LIN {X 0,Y 523.916,Z 196.85,A -85,B 0,C 180,E1 -4806.403,E2 -4806.403} C_VEL
LIN {X 0,Y 523.927,Z 196.844,A -85,B 0,C 180,E1 -4809.083,E2 -4809.083} C_VEL
LIN {X 0,Y 523.968,Z 196.839,A -85,B 0,C 180,E1 -4811.312,E2 -4811.312} C_VEL
LIN {X 0,Y 523.951,Z 196.84,A -85,B 0,C 180,E1 -4814.691,E2 -4814.691} C_VEL
LIN {X 0,Y 523.951,Z 196.846,A -85,B 0,C 180,E1 -4817.881,E2 -4817.881} C_VEL
LIN {X 0,Y 523.972,Z 196.843,A -85,B 0,C 180,E1 -4819.923,E2 -4819.923} C_VEL
LIN {X 0,Y 523.905,Z 196.844,A -85,B 0,C 180,E1 -4822.868,E2 -4822.868} C_VEL
LIN {X 0,Y 523.937,Z 196.847,A -85,B 0,C 180,E1 -4825.71,E2 -4825.71} C_VEL
LIN {X 0,Y 523.925,Z 196.843,A -85,B 0,C 180,E1 -4828.456,E2 -4828.456} C_VEL
LIN {X 0,Y 523.943,Z 196.841,A -85,B 0,C 180,E1 -4831.126,E2 -4831.126} C_VEL
LIN {X 0,Y 523.975,Z 196.842,A -85,B 0,C 180,E1 -4833.98,E2 -4833.98} C_VEL
LIN {X 0,Y 523.928,Z 196.842,A -85,B 0,C 180,E1 -4836.27,E2 -4836.27} C_VEL
LIN {X 0,Y 523.938,Z 196.834,A -85,B 0,C 180,E1 -4838.766,E2 -4838.766} C_VEL
LIN {X 0,Y 523.945,Z 196.843,A -85,B 0,C 180,E1 -4841.221,E2 -4841.221} C_VEL
LIN {X 0,Y 523.932,Z 196.848,A -85,B 0,C 180,E1 -4843.639,E2 -4843.639} C_VEL
LIN {X 0,Y 523.932,Z 196.844,A -85,B 0,C 180,E1 -4846.028,E2 -4846.028} C_VEL
LIN {X 0,Y 524.002,Z 196.833,A -85,B 0,C 180,E1 -4848.394,E2 -4848.394} C_VEL
LIN {X 0,Y 523.999,Z 196.84,A -85,B 0,C 180,E1 -4851.516,E2 -4851.516} C_VEL
LIN {X 0,Y 524.077,Z 196.824,A -85,B 0,C 180,E1 -4854.614,E2 -4854.614} C_VEL
LIN {X 0,Y 524.102,Z 196.826,A -85,B 0,C 180,E1 -4857.695,E2 -4857.695} C_VEL
LIN {X 0,Y 524.117,Z 196.818,A -85,B 0,C 180,E1 -4860.768,E2 -4860.768} C_VEL
LIN {X 0,Y 524.067,Z 196.83,A -85,B 0,C 180,E1 -4863.075,E2 -4863.075} C_VEL
LIN {X 0,Y 524.037,Z 196.829,A -85,B 0,C 180,E1 -4866.159,E2 -4866.159} C_VEL
LIN {X 0,Y 523.995,Z 196.84,A -85,B 0,C 180,E1 -4869.262,E2 -4869.262} C_VEL
LIN {X 0,Y 523.999,Z 196.835,A -85,B 0,C 180,E1 -4871.743,E2 -4871.743} C_VEL
LIN {X 0,Y 523.983,Z 196.843,A -85,B 0,C 180,E1 -4875.053,E2 -4875.053} C_VEL
LIN {X 0,Y 523.956,Z 196.839,A -85,B 0,C 180,E1 -4877.969,E2 -4877.969} C_VEL
LIN {X 0,Y 523.963,Z 196.838,A -85,B 0,C 180,E1 -4880.41,E2 -4880.41} C_VEL
LIN {X 0,Y 523.908,Z 196.851,A -85,B 0,C 180,E1 -4882.894,E2 -4882.894} C_VEL
LIN {X 0,Y 523.945,Z 196.835,A -85,B 0,C 180,E1 -4885.419,E2 -4885.419} C_VEL
LIN {X 0,Y 523.963,Z 196.837,A -85,B 0,C 180,E1 -4887.999,E2 -4887.999} C_VEL
LIN {X 0,Y 523.946,Z 196.847,A -85,B 0,C 180,E1 -4890.857,E2 -4890.857} C_VEL
LIN {X 0,Y 523.955,Z 196.838,A -85,B 0,C 180,E1 -4893.736,E2 -4893.736} C_VEL
LIN {X 0,Y 523.917,Z 196.846,A -85,B 0,C 180,E1 -4896.405,E2 -4896.405} C_VEL
LIN {X 0,Y 523.918,Z 196.848,A -85,B 0,C 180,E1 -4899.085,E2 -4899.085} C_VEL
LIN {X 0,Y 523.951,Z 196.839,A -85,B 0,C 180,E1 -4902.119,E2 -4902.119} C_VEL
LIN {X 0,Y 523.951,Z 196.842,A -85,B 0,C 180,E1 -4905.309,E2 -4905.309} C_VEL
LIN {X 0,Y 523.919,Z 196.851,A -85,B 0,C 180,E1 -4906.923,E2 -4906.923} C_VEL
LIN {X 0,Y 523.252,Z 196.929,A -85,B 0,C 180,E1 -4907.564,E2 -4907.564} C_VEL
LIN {X 0,Y 520.407,Z 197.288,A -85,B 0,C 180,E1 -4908.606,E2 -4908.606} C_VEL
LIN {X 0,Y 518.001,Z 197.588,A -85,B 0,C 180,E1 -4909.445,E2 -4909.445} C_VEL
LIN {X 0,Y 516.964,Z 197.715,A -85,B 0,C 180,E1 -4910.093,E2 -4910.093} C_VEL
LIN {X 0,Y 516.878,Z 197.725,A -85,B 0,C 180,E1 -4910.312,E2 -4910.312} C_VEL
LIN {X 0,Y 516.874,Z 197.722,A -85,B 0,C 180,E1 -4913.344,E2 -4913.344} C_VEL
LIN {X 0,Y 516.905,Z 197.721,A -85,B 0,C 180,E1 -4916.121,E2 -4916.121} C_VEL
LIN {X 0,Y 516.89,Z 197.725,A -85,B 0,C 180,E1 -4918.936,E2 -4918.936} C_VEL
LIN {X 0,Y 516.918,Z 197.719,A -85,B 0,C 180,E1 -4921.585,E2 -4921.585} C_VEL
LIN {X 0,Y 516.91,Z 197.725,A -85,B 0,C 180,E1 -4924.642,E2 -4924.642} C_VEL
LIN {X 0,Y 516.927,Z 197.807,A -85,B 0,C 180,E1 -4924.939,E2 -4924.939} C_VEL
LIN {X 0,Y 519.115,Z 207.96,A -85,B 0,C 180,E1 -4926.672,E2 -4926.672} C_VEL
LIN {X 0,Y 518.935,Z 218.424,A -85,B 0,C 180,E1 -4928.27,E2 -4928.27} C_VEL
LIN {X 0,Y 521.961,Z 232.108,A -85,B 0,C 180,E1 -4928.602,E2 -4928.602} C_VEL
LIN {X 0,Y 520.964,Z 381.412,A -85,B 0,C 180,E1 -4930.729,E2 -4930.729} C_VEL
LIN {X 0,Y 520.722,Z 395.433,A -85,B 0,C 180,E1 -4931.049,E2 -4931.049} C_VEL
LIN {X 0,Y 520.379,Z 409.153,A -85,B 0,C 180,E1 -4931.496,E2 -4931.496} C_VEL
LIN {X 0,Y 519.89,Z 422.978,A -85,B 0,C 180,E1 -4932.089,E2 -4932.089} C_VEL
LIN {X 0,Y 519.503,Z 435.806,A -85,B 0,C 180,E1 -4932.787,E2 -4932.787} C_VEL
LIN {X 0,Y 518.969,Z 449.181,A -85,B 0,C 180,E1 -4933.681,E2 -4933.681} C_VEL
LIN {X 0,Y 518.45,Z 461.571,A -85,B 0,C 180,E1 -4934.687,E2 -4934.687} C_VEL
LIN {X 0,Y 517.921,Z 473.611,A -85,B 0,C 180,E1 -4935.863,E2 -4935.863} C_VEL
LIN {X 0,Y 517.492,Z 483.799,A -85,B 0,C 180,E1 -4937.051,E2 -4937.051} C_VEL
LIN {X 0,Y 517.082,Z 493.77,A -85,B 0,C 180,E1 -4938.435,E2 -4938.435} C_VEL
LIN {X 0,Y 516.807,Z 502.039,A -85,B 0,C 180,E1 -4939.818,E2 -4939.818} C_VEL
LIN {X 0,Y 516.575,Z 509.804,A -85,B 0,C 180,E1 -4941.393,E2 -4941.393} C_VEL
LIN {X 0,Y 516.408,Z 515.988,A -85,B 0,C 180,E1 -4942.965,E2 -4942.965} C_VEL
LIN {X 0,Y 516.383,Z 520.763,A -85,B 0,C 180,E1 -4944.533,E2 -4944.533} C_VEL
LIN {X 0,Y 516.326,Z 524.265,A -85,B 0,C 180,E1 -4946.098,E2 -4946.098} C_VEL
LIN {X 0,Y 516.259,Z 526.586,A -85,B 0,C 180,E1 -4947.659,E2 -4947.659} C_VEL
LIN {X 0,Y 516.156,Z 527.776,A -85,B 0,C 180,E1 -4949.22,E2 -4949.22} C_VEL
LIN {X 0,Y 516.157,Z 527.795,A -85,B 0,C 180,E1 -4950.78,E2 -4950.78} C_VEL
LIN {X 0,Y 516.259,Z 526.681,A -85,B 0,C 180,E1 -4952.341,E2 -4952.341} C_VEL
LIN {X 0,Y 516.326,Z 524.436,A -85,B 0,C 180,E1 -4953.902,E2 -4953.902} C_VEL
LIN {X 0,Y 516.379,Z 521.005,A -85,B 0,C 180,E1 -4955.467,E2 -4955.467} C_VEL
LIN {X 0,Y 516.407,Z 516.308,A -85,B 0,C 180,E1 -4957.035,E2 -4957.035} C_VEL
LIN {X 0,Y 516.573,Z 510.218,A -85,B 0,C 180,E1 -4958.607,E2 -4958.607} C_VEL
LIN {X 0,Y 516.802,Z 502.549,A -85,B 0,C 180,E1 -4960.182,E2 -4960.182} C_VEL
LIN {X 0,Y 517.064,Z 494.37,A -85,B 0,C 180,E1 -4961.565,E2 -4961.565} C_VEL
LIN {X 0,Y 517.453,Z 484.518,A -85,B 0,C 180,E1 -4962.95,E2 -4962.95} C_VEL
LIN {X 0,Y 517.887,Z 474.412,A -85,B 0,C 180,E1 -4964.138,E2 -4964.138} C_VEL
LIN {X 0,Y 518.366,Z 462.579,A -85,B 0,C 180,E1 -4965.311,E2 -4965.311} C_VEL
LIN {X 0,Y 518.917,Z 450.576,A -85,B 0,C 180,E1 -4966.301,E2 -4966.301} C_VEL
LIN {X 0,Y 519.386,Z 438.788,A -85,B 0,C 180,E1 -4967.116,E2 -4967.116} C_VEL
LIN {X 0,Y 519.863,Z 424.732,A -85,B 0,C 180,E1 -4967.912,E2 -4967.912} C_VEL
LIN {X 0,Y 520.353,Z 410.13,A -85,B 0,C 180,E1 -4968.556,E2 -4968.556} C_VEL
LIN {X 0,Y 520.665,Z 394.698,A -85,B 0,C 180,E1 -4969.063,E2 -4969.063} C_VEL
LIN {X 0,Y 520.953,Z 379.884,A -85,B 0,C 180,E1 -4969.388,E2 -4969.388} C_VEL
LIN {X 0,Y 521.999,Z 232.476,A -85,B 0,C 180,E1 -4971.481,E2 -4971.481} C_VEL
LIN {X 0,Y 518.886,Z 218.209,A -85,B 0,C 180,E1 -4971.828,E2 -4971.828} C_VEL
LIN {X 0,Y 519.197,Z 208.527,A -85,B 0,C 180,E1 -4973.324,E2 -4973.324} C_VEL
LIN {X 0,Y 516.932,Z 197.723,A -85,B 0,C 180,E1 -4975.195,E2 -4975.195} C_VEL
LIN {X 0,Y 516.926,Z 197.722,A -85,B 0,C 180,E1 -4977.905,E2 -4977.905} C_VEL
LIN {X 0,Y 516.891,Z 197.722,A -85,B 0,C 180,E1 -4980.203,E2 -4980.203} C_VEL
LIN {X 0,Y 516.895,Z 197.723,A -85,B 0,C 180,E1 -4982.946,E2 -4982.946} C_VEL
LIN {X 0,Y 516.884,Z 197.725,A -85,B 0,C 180,E1 -4985.778,E2 -4985.778} C_VEL
LIN {X 0,Y 516.879,Z 197.724,A -85,B 0,C 180,E1 -4988.715,E2 -4988.715} C_VEL
LIN {X 0,Y 516.912,Z 197.72,A -85,B 0,C 180,E1 -4991.774,E2 -4991.774} C_VEL
LIN {X 0,Y 516.918,Z 197.72,A -85,B 0,C 180,E1 -4995.009,E2 -4995.009} C_VEL
LIN {X 0,Y 516.917,Z 197.713,A -85,B 0,C 180,E1 -4998.397,E2 -4998.397} C_VEL
LIN {X 0,Y 516.877,Z 197.724,A -85,B 0,C 180,E1 -5001.284,E2 -5001.284} C_VEL
LIN {X 0,Y 516.885,Z 197.719,A -85,B 0,C 180,E1 -5004.221,E2 -5004.221} C_VEL
LIN {X 0,Y 516.891,Z 197.723,A -85,B 0,C 180,E1 -5007.053,E2 -5007.053} C_VEL
LIN {X 0,Y 516.895,Z 197.717,A -85,B 0,C 180,E1 -5009.796,E2 -5009.796} C_VEL
LIN {X 0,Y 516.921,Z 197.717,A -85,B 0,C 180,E1 -5012.467,E2 -5012.467} C_VEL
LIN {X 0,Y 516.902,Z 197.726,A -85,B 0,C 180,E1 -5015.071,E2 -5015.071} C_VEL
LIN {X 0,Y 516.878,Z 197.722,A -85,B 0,C 180,E1 -5018.462,E2 -5018.462} C_VEL
LIN {X 0,Y 516.897,Z 197.724,A -85,B 0,C 180,E1 -5020.955,E2 -5020.955} C_VEL
LIN {X 0,Y 516.909,Z 197.719,A -85,B 0,C 180,E1 -5023.41,E2 -5023.41} C_VEL
LIN {X 0,Y 516.886,Z 197.717,A -85,B 0,C 180,E1 -5025.833,E2 -5025.833} C_VEL
LIN {X 0,Y 516.956,Z 197.713,A -85,B 0,C 180,E1 -5028.233,E2 -5028.233} C_VEL
LIN {X 0,Y 516.961,Z 197.712,A -85,B 0,C 180,E1 -5031.399,E2 -5031.399} C_VEL
LIN {X 0,Y 517.001,Z 197.704,A -85,B 0,C 180,E1 -5033.757,E2 -5033.757} C_VEL
LIN {X 0,Y 517.007,Z 197.711,A -85,B 0,C 180,E1 -5036.883,E2 -5036.883} C_VEL
LIN {X 0,Y 517.073,Z 197.695,A -85,B 0,C 180,E1 -5040,E2 -5040} C_VEL
LIN {X 0,Y 517.008,Z 197.705,A -85,B 0,C 180,E1 -5043.117,E2 -5043.117} C_VEL
LIN {X 0,Y 517,Z 197.71,A -85,B 0,C 180,E1 -5046.243,E2 -5046.243} C_VEL
LIN {X 0,Y 516.949,Z 197.711,A -85,B 0,C 180,E1 -5049.389,E2 -5049.389} C_VEL
LIN {X 0,Y 516.947,Z 197.713,A -85,B 0,C 180,E1 -5051.81,E2 -5051.81} C_VEL
LIN {X 0,Y 516.937,Z 197.715,A -85,B 0,C 180,E1 -5055.148,E2 -5055.148} C_VEL
LIN {X 0,Y 516.917,Z 197.72,A -85,B 0,C 180,E1 -5058.222,E2 -5058.222} C_VEL
LIN {X 0,Y 516.904,Z 197.72,A -85,B 0,C 180,E1 -5060.702,E2 -5060.702} C_VEL
LIN {X 0,Y 516.902,Z 197.724,A -85,B 0,C 180,E1 -5064.072,E2 -5064.072} C_VEL
LIN {X 0,Y 516.918,Z 197.72,A -85,B 0,C 180,E1 -5066.658,E2 -5066.658} C_VEL
LIN {X 0,Y 516.917,Z 197.717,A -85,B 0,C 180,E1 -5069.527,E2 -5069.527} C_VEL
LIN {X 0,Y 516.893,Z 197.721,A -85,B 0,C 180,E1 -5072.545,E2 -5072.545} C_VEL
LIN {X 0,Y 516.876,Z 197.721,A -85,B 0,C 180,E1 -5075.333,E2 -5075.333} C_VEL
LIN {X 0,Y 516.874,Z 197.727,A -85,B 0,C 180,E1 -5077.944,E2 -5077.944} C_VEL
LIN {X 0,Y 516.879,Z 197.717,A -85,B 0,C 180,E1 -5080.742,E2 -5080.742} C_VEL
LIN {X 0,Y 516.878,Z 197.722,A -85,B 0,C 180,E1 -5082.832,E2 -5082.832} C_VEL
LIN {X 0,Y 516.917,Z 197.717,A -85,B 0,C 180,E1 -5085.011,E2 -5085.011} C_VEL
LIN {X 0,Y 516.918,Z 197.719,A -85,B 0,C 180,E1 -5088.398,E2 -5088.398} C_VEL
LIN {X 0,Y 516.882,Z 197.722,A -85,B 0,C 180,E1 -5091.285,E2 -5091.285} C_VEL
LIN {X 0,Y 516.884,Z 197.726,A -85,B 0,C 180,E1 -5094.222,E2 -5094.222} C_VEL
LIN {X 0,Y 516.893,Z 197.721,A -85,B 0,C 180,E1 -5097.054,E2 -5097.054} C_VEL
LIN {X 0,Y 516.889,Z 197.727,A -85,B 0,C 180,E1 -5099.797,E2 -5099.797} C_VEL
LIN {X 0,Y 516.942,Z 197.766,A -85,B 0,C 180,E1 -5101.726,E2 -5101.726} C_VEL
LIN {X 0,Y 519.956,Z 211.044,A -85,B 0,C 180,E1 -5103.727,E2 -5103.727} C_VEL
LIN {X 0,Y 519.317,Z 231.522,A -85,B 0,C 180,E1 -5106.471,E2 -5106.471} C_VEL
LIN {X 0,Y 518.882,Z 244.581,A -85,B 0,C 180,E1 -5108.199,E2 -5108.199} C_VEL
LIN {X 0,Y 521.857,Z 259.942,A -85,B 0,C 180,E1 -5108.558,E2 -5108.558} C_VEL
LIN {X 0,Y 520.958,Z 393.454,A -85,B 0,C 180,E1 -5110.442,E2 -5110.442} C_VEL
LIN {X 0,Y 520.783,Z 413.905,A -85,B 0,C 180,E1 -5110.772,E2 -5110.772} C_VEL
LIN {X 0,Y 520.463,Z 428.98,A -85,B 0,C 180,E1 -5111.167,E2 -5111.167} C_VEL
LIN {X 0,Y 520.064,Z 443.174,A -85,B 0,C 180,E1 -5111.688,E2 -5111.688} C_VEL
LIN {X 0,Y 519.498,Z 457.644,A -85,B 0,C 180,E1 -5112.381,E2 -5112.381} C_VEL
LIN {X 0,Y 519.055,Z 470.865,A -85,B 0,C 180,E1 -5113.177,E2 -5113.177} C_VEL
LIN {X 0,Y 518.569,Z 483.587,A -85,B 0,C 180,E1 -5114.11,E2 -5114.11} C_VEL
LIN {X 0,Y 517.958,Z 496.586,A -85,B 0,C 180,E1 -5115.262,E2 -5115.262} C_VEL
LIN {X 0,Y 517.529,Z 507.783,A -85,B 0,C 180,E1 -5116.453,E2 -5116.453} C_VEL
LIN {X 0,Y 517.131,Z 518.653,A -85,B 0,C 180,E1 -5117.84,E2 -5117.84} C_VEL
LIN {X 0,Y 516.865,Z 527.703,A -85,B 0,C 180,E1 -5119.225,E2 -5119.225} C_VEL
LIN {X 0,Y 516.575,Z 535.208,A -85,B 0,C 180,E1 -5120.604,E2 -5120.604} C_VEL
LIN {X 0,Y 516.443,Z 542.215,A -85,B 0,C 180,E1 -5122.179,E2 -5122.179} C_VEL
LIN {X 0,Y 516.36,Z 547.724,A -85,B 0,C 180,E1 -5123.749,E2 -5123.749} C_VEL
LIN {X 0,Y 516.238,Z 551.887,A -85,B 0,C 180,E1 -5125.315,E2 -5125.315} C_VEL
LIN {X 0,Y 516.271,Z 554.808,A -85,B 0,C 180,E1 -5126.879,E2 -5126.879} C_VEL
LIN {X 0,Y 516.189,Z 556.548,A -85,B 0,C 180,E1 -5128.44,E2 -5128.44} C_VEL
LIN {X 0,Y 516.151,Z 557.144,A -85,B 0,C 180,E1 -5130,E2 -5130} C_VEL
LIN {X 0,Y 516.189,Z 556.545,A -85,B 0,C 180,E1 -5131.56,E2 -5131.56} C_VEL
LIN {X 0,Y 516.271,Z 554.803,A -85,B 0,C 180,E1 -5133.121,E2 -5133.121} C_VEL
LIN {X 0,Y 516.238,Z 551.885,A -85,B 0,C 180,E1 -5134.685,E2 -5134.685} C_VEL
LIN {X 0,Y 516.375,Z 547.728,A -85,B 0,C 180,E1 -5136.251,E2 -5136.251} C_VEL
LIN {X 0,Y 516.443,Z 542.216,A -85,B 0,C 180,E1 -5137.821,E2 -5137.821} C_VEL
LIN {X 0,Y 516.575,Z 535.202,A -85,B 0,C 180,E1 -5139.396,E2 -5139.396} C_VEL
LIN {X 0,Y 516.863,Z 527.698,A -85,B 0,C 180,E1 -5140.775,E2 -5140.775} C_VEL
LIN {X 0,Y 517.097,Z 518.923,A -85,B 0,C 180,E1 -5142.121,E2 -5142.121} C_VEL
LIN {X 0,Y 517.489,Z 509.423,A -85,B 0,C 180,E1 -5143.348,E2 -5143.348} C_VEL
LIN {X 0,Y 517.917,Z 498.552,A -85,B 0,C 180,E1 -5144.539,E2 -5144.539} C_VEL
LIN {X 0,Y 518.355,Z 487.283,A -85,B 0,C 180,E1 -5145.582,E2 -5145.582} C_VEL
LIN {X 0,Y 518.912,Z 473.727,A -85,B 0,C 180,E1 -5146.625,E2 -5146.625} C_VEL
LIN {X 0,Y 519.493,Z 459.409,A -85,B 0,C 180,E1 -5147.518,E2 -5147.518} C_VEL
LIN {X 0,Y 519.957,Z 445.443,A -85,B 0,C 180,E1 -5148.214,E2 -5148.214} C_VEL
LIN {X 0,Y 520.407,Z 430.524,A -85,B 0,C 180,E1 -5148.784,E2 -5148.784} C_VEL
LIN {X 0,Y 520.758,Z 415.339,A -85,B 0,C 180,E1 -5149.197,E2 -5149.197} C_VEL
LIN {X 0,Y 520.972,Z 395.646,A -85,B 0,C 180,E1 -5149.526,E2 -5149.526} C_VEL
LIN {X 0,Y 521.861,Z 259.839,A -85,B 0,C 180,E1 -5151.443,E2 -5151.443} C_VEL
LIN {X 0,Y 518.886,Z 244.592,A -85,B 0,C 180,E1 -5151.799,E2 -5151.799} C_VEL
LIN {X 0,Y 519.653,Z 222.079,A -85,B 0,C 180,E1 -5154.787,E2 -5154.787} C_VEL
LIN {X 0,Y 519.956,Z 211.043,A -85,B 0,C 180,E1 -5156.273,E2 -5156.273} C_VEL
LIN {X 0,Y 516.919,Z 197.724,A -85,B 0,C 180,E1 -5158.31,E2 -5158.31} C_VEL
LIN {X 0,Y 516.886,Z 197.719,A -85,B 0,C 180,E1 -5161.109,E2 -5161.109} C_VEL
LIN {X 0,Y 516.908,Z 197.718,A -85,B 0,C 180,E1 -5163.966,E2 -5163.966} C_VEL
LIN {X 0,Y 516.878,Z 197.723,A -85,B 0,C 180,E1 -5166.745,E2 -5166.745} C_VEL
LIN {X 0,Y 516.899,Z 197.724,A -85,B 0,C 180,E1 -5169.719,E2 -5169.719} C_VEL
LIN {X 0,Y 516.914,Z 197.722,A -85,B 0,C 180,E1 -5171.774,E2 -5171.774} C_VEL
LIN {X 0,Y 516.917,Z 197.715,A -85,B 0,C 180,E1 -5175.009,E2 -5175.009} C_VEL
LIN {X 0,Y 516.916,Z 197.718,A -85,B 0,C 180,E1 -5178.397,E2 -5178.397} C_VEL
LIN {X 0,Y 516.88,Z 197.721,A -85,B 0,C 180,E1 -5181.284,E2 -5181.284} C_VEL
LIN {X 0,Y 516.884,Z 197.722,A -85,B 0,C 180,E1 -5184.221,E2 -5184.221} C_VEL
LIN {X 0,Y 516.89,Z 197.717,A -85,B 0,C 180,E1 -5187.053,E2 -5187.053} C_VEL
LIN {X 0,Y 516.894,Z 197.724,A -85,B 0,C 180,E1 -5189.797,E2 -5189.797} C_VEL
LIN {X 0,Y 516.92,Z 197.715,A -85,B 0,C 180,E1 -5192.467,E2 -5192.467} C_VEL
LIN {X 0,Y 516.902,Z 197.719,A -85,B 0,C 180,E1 -5195.072,E2 -5195.072} C_VEL
LIN {X 0,Y 516.878,Z 197.713,A -85,B 0,C 180,E1 -5198.462,E2 -5198.462} C_VEL
LIN {X 0,Y 516.896,Z 197.718,A -85,B 0,C 180,E1 -5200.955,E2 -5200.955} C_VEL
LIN {X 0,Y 516.909,Z 197.723,A -85,B 0,C 180,E1 -5203.41,E2 -5203.41} C_VEL
LIN {X 0,Y 516.887,Z 197.724,A -85,B 0,C 180,E1 -5205.833,E2 -5205.833} C_VEL
LIN {X 0,Y 516.948,Z 197.714,A -85,B 0,C 180,E1 -5209.028,E2 -5209.028} C_VEL
LIN {X 0,Y 516.969,Z 197.709,A -85,B 0,C 180,E1 -5212.187,E2 -5212.187} C_VEL
LIN {X 0,Y 517.024,Z 197.702,A -85,B 0,C 180,E1 -5214.54,E2 -5214.54} C_VEL
LIN {X 0,Y 517.074,Z 197.702,A -85,B 0,C 180,E1 -5217.663,E2 -5217.663} C_VEL
LIN {X 0,Y 517.087,Z 197.694,A -85,B 0,C 180,E1 -5220.779,E2 -5220.779} C_VEL
LIN {X 0,Y 517.008,Z 197.71,A -85,B 0,C 180,E1 -5223.117,E2 -5223.117} C_VEL
LIN {X 0,Y 517.001,Z 197.705,A -85,B 0,C 180,E1 -5226.243,E2 -5226.243} C_VEL
LIN {X 0,Y 516.949,Z 197.719,A -85,B 0,C 180,E1 -5229.389,E2 -5229.389} C_VEL
LIN {X 0,Y 516.948,Z 197.712,A -85,B 0,C 180,E1 -5231.811,E2 -5231.811} C_VEL
LIN {X 0,Y 516.935,Z 197.722,A -85,B 0,C 180,E1 -5235.147,E2 -5235.147} C_VEL
LIN {X 0,Y 516.917,Z 197.716,A -85,B 0,C 180,E1 -5238.223,E2 -5238.223} C_VEL
LIN {X 0,Y 516.904,Z 197.72,A -85,B 0,C 180,E1 -5240.702,E2 -5240.702} C_VEL
LIN {X 0,Y 516.903,Z 197.716,A -85,B 0,C 180,E1 -5244.073,E2 -5244.073} C_VEL
LIN {X 0,Y 516.919,Z 197.71,A -85,B 0,C 180,E1 -5246.658,E2 -5246.658} C_VEL
LIN {X 0,Y 516.918,Z 197.718,A -85,B 0,C 180,E1 -5249.527,E2 -5249.527} C_VEL
LIN {X 0,Y 516.894,Z 197.722,A -85,B 0,C 180,E1 -5252.545,E2 -5252.545} C_VEL
LIN {X 0,Y 516.877,Z 197.724,A -85,B 0,C 180,E1 -5255.333,E2 -5255.333} C_VEL
LIN {X 0,Y 516.876,Z 197.72,A -85,B 0,C 180,E1 -5257.944,E2 -5257.944} C_VEL
LIN {X 0,Y 516.88,Z 197.727,A -85,B 0,C 180,E1 -5260.742,E2 -5260.742} C_VEL
LIN {X 0,Y 516.898,Z 197.726,A -85,B 0,C 180,E1 -5262.83,E2 -5262.83} C_VEL
LIN {X 0,Y 516.918,Z 197.721,A -85,B 0,C 180,E1 -5265.011,E2 -5265.011} C_VEL
LIN {X 0,Y 516.913,Z 197.721,A -85,B 0,C 180,E1 -5268.399,E2 -5268.399} C_VEL
LIN {X 0,Y 516.878,Z 197.725,A -85,B 0,C 180,E1 -5270.312,E2 -5270.312} C_VEL
LIN {X 0,Y 516.207,Z 197.808,A -85,B 0,C 180,E1 -5270.962,E2 -5270.962} C_VEL
LIN {X 0,Y 513.36,Z 198.16,A -85,B 0,C 180,E1 -5272.018,E2 -5272.018} C_VEL
LIN {X 0,Y 510.949,Z 198.466,A -85,B 0,C 180,E1 -5272.868,E2 -5272.868} C_VEL
LIN {X 0,Y 509.906,Z 198.59,A -85,B 0,C 180,E1 -5273.525,E2 -5273.525} C_VEL
LIN {X 0,Y 509.817,Z 198.6,A -85,B 0,C 180,E1 -5273.747,E2 -5273.747} C_VEL
LIN {X 0,Y 509.857,Z 198.601,A -85,B 0,C 180,E1 -5276.54,E2 -5276.54} C_VEL
LIN {X 0,Y 509.844,Z 198.601,A -85,B 0,C 180,E1 -5279.335,E2 -5279.335} C_VEL
LIN {X 0,Y 509.893,Z 198.597,A -85,B 0,C 180,E1 -5282.055,E2 -5282.055} C_VEL
LIN {X 0,Y 509.872,Z 198.661,A -85,B 0,C 180,E1 -5284.677,E2 -5284.677} C_VEL
LIN {X 0,Y 512.223,Z 209.489,A -85,B 0,C 180,E1 -5286.554,E2 -5286.554} C_VEL
LIN {X 0,Y 512.076,Z 218.377,A -85,B 0,C 180,E1 -5287.952,E2 -5287.952} C_VEL
LIN {X 0,Y 515.356,Z 232.894,A -85,B 0,C 180,E1 -5288.322,E2 -5288.322} C_VEL
LIN {X 0,Y 514.284,Z 379.059,A -85,B 0,C 180,E1 -5290.423,E2 -5290.423} C_VEL
LIN {X 0,Y 514.013,Z 394.613,A -85,B 0,C 180,E1 -5290.762,E2 -5290.762} C_VEL
LIN {X 0,Y 513.657,Z 409.37,A -85,B 0,C 180,E1 -5291.245,E2 -5291.245} C_VEL
LIN {X 0,Y 513.127,Z 423.191,A -85,B 0,C 180,E1 -5291.845,E2 -5291.845} C_VEL
LIN {X 0,Y 512.724,Z 436.017,A -85,B 0,C 180,E1 -5292.552,E2 -5292.552} C_VEL
LIN {X 0,Y 512.126,Z 449.391,A -85,B 0,C 180,E1 -5293.456,E2 -5293.456} C_VEL
LIN {X 0,Y 511.566,Z 462.071,A -85,B 0,C 180,E1 -5294.502,E2 -5294.502} C_VEL
LIN {X 0,Y 510.985,Z 473.82,A -85,B 0,C 180,E1 -5295.667,E2 -5295.667} C_VEL
LIN {X 0,Y 510.552,Z 484.006,A -85,B 0,C 180,E1 -5296.872,E2 -5296.872} C_VEL
LIN {X 0,Y 510.07,Z 494.421,A -85,B 0,C 180,E1 -5298.341,E2 -5298.341} C_VEL
LIN {X 0,Y 509.743,Z 503.337,A -85,B 0,C 180,E1 -5299.876,E2 -5299.876} C_VEL
LIN {X 0,Y 509.515,Z 510.009,A -85,B 0,C 180,E1 -5301.273,E2 -5301.273} C_VEL
LIN {X 0,Y 509.356,Z 516.191,A -85,B 0,C 180,E1 -5302.867,E2 -5302.867} C_VEL
LIN {X 0,Y 509.323,Z 520.965,A -85,B 0,C 180,E1 -5304.457,E2 -5304.457} C_VEL
LIN {X 0,Y 509.252,Z 524.467,A -85,B 0,C 180,E1 -5306.043,E2 -5306.043} C_VEL
LIN {X 0,Y 509.187,Z 526.786,A -85,B 0,C 180,E1 -5307.627,E2 -5307.627} C_VEL
LIN {X 0,Y 509.07,Z 527.977,A -85,B 0,C 180,E1 -5309.209,E2 -5309.209} C_VEL
LIN {X 0,Y 509.071,Z 527.996,A -85,B 0,C 180,E1 -5310.791,E2 -5310.791} C_VEL
LIN {X 0,Y 509.188,Z 526.881,A -85,B 0,C 180,E1 -5312.373,E2 -5312.373} C_VEL
LIN {X 0,Y 509.252,Z 524.635,A -85,B 0,C 180,E1 -5313.957,E2 -5313.957} C_VEL
LIN {X 0,Y 509.317,Z 521.204,A -85,B 0,C 180,E1 -5315.543,E2 -5315.543} C_VEL
LIN {X 0,Y 509.356,Z 516.506,A -85,B 0,C 180,E1 -5317.133,E2 -5317.133} C_VEL
LIN {X 0,Y 509.513,Z 510.417,A -85,B 0,C 180,E1 -5318.727,E2 -5318.727} C_VEL
LIN {X 0,Y 509.788,Z 502.747,A -85,B 0,C 180,E1 -5320.324,E2 -5320.324} C_VEL
LIN {X 0,Y 510.064,Z 494.159,A -85,B 0,C 180,E1 -5321.789,E2 -5321.789} C_VEL
LIN {X 0,Y 510.524,Z 484.714,A -85,B 0,C 180,E1 -5323.129,E2 -5323.129} C_VEL
LIN {X 0,Y 510.973,Z 474.608,A -85,B 0,C 180,E1 -5324.334,E2 -5324.334} C_VEL
LIN {X 0,Y 511.489,Z 463.047,A -85,B 0,C 180,E1 -5325.496,E2 -5325.496} C_VEL
LIN {X 0,Y 512.09,Z 450.515,A -85,B 0,C 180,E1 -5326.545,E2 -5326.545} C_VEL
LIN {X 0,Y 512.695,Z 437.402,A -85,B 0,C 180,E1 -5327.449,E2 -5327.449} C_VEL
LIN {X 0,Y 513.108,Z 424.921,A -85,B 0,C 180,E1 -5328.156,E2 -5328.156} C_VEL
LIN {X 0,Y 513.625,Z 410.315,A -85,B 0,C 180,E1 -5328.808,E2 -5328.808} C_VEL
LIN {X 0,Y 513.97,Z 394.993,A -85,B 0,C 180,E1 -5329.318,E2 -5329.318} C_VEL
LIN {X 0,Y 514.285,Z 379.346,A -85,B 0,C 180,E1 -5329.662,E2 -5329.662} C_VEL
LIN {X 0,Y 515.341,Z 232.959,A -85,B 0,C 180,E1 -5331.767,E2 -5331.767} C_VEL
LIN {X 0,Y 512.076,Z 218.337,A -85,B 0,C 180,E1 -5332.143,E2 -5332.143} C_VEL
LIN {X 0,Y 512.323,Z 210.046,A -85,B 0,C 180,E1 -5333.441,E2 -5333.441} C_VEL
LIN {X 0,Y 509.869,Z 198.603,A -85,B 0,C 180,E1 -5335.46,E2 -5335.46} C_VEL
LIN {X 0,Y 509.897,Z 198.596,A -85,B 0,C 180,E1 -5338.1,E2 -5338.1} C_VEL
LIN {X 0,Y 509.844,Z 198.605,A -85,B 0,C 180,E1 -5341.279,E2 -5341.279} C_VEL
LIN {X 0,Y 509.858,Z 198.598,A -85,B 0,C 180,E1 -5344.202,E2 -5344.202} C_VEL
LIN {X 0,Y 509.816,Z 198.607,A -85,B 0,C 180,E1 -5347.34,E2 -5347.34} C_VEL
LIN {X 0,Y 509.835,Z 198.598,A -85,B 0,C 180,E1 -5350.381,E2 -5350.381} C_VEL
LIN {X 0,Y 509.836,Z 198.603,A -85,B 0,C 180,E1 -5353.064,E2 -5353.064} C_VEL
LIN {X 0,Y 509.826,Z 198.601,A -85,B 0,C 180,E1 -5355.792,E2 -5355.792} C_VEL
LIN {X 0,Y 509.86,Z 198.593,A -85,B 0,C 180,E1 -5358.575,E2 -5358.575} C_VEL
LIN {X 0,Y 509.846,Z 198.593,A -85,B 0,C 180,E1 -5361.786,E2 -5361.786} C_VEL
LIN {X 0,Y 509.84,Z 198.598,A -85,B 0,C 180,E1 -5364.623,E2 -5364.623} C_VEL
LIN {X 0,Y 509.859,Z 198.592,A -85,B 0,C 180,E1 -5367.481,E2 -5367.481} C_VEL
LIN {X 0,Y 509.875,Z 198.591,A -85,B 0,C 180,E1 -5370.268,E2 -5370.268} C_VEL
LIN {X 0,Y 509.878,Z 198.6,A -85,B 0,C 180,E1 -5372.944,E2 -5372.944} C_VEL
LIN {X 0,Y 509.861,Z 198.597,A -85,B 0,C 180,E1 -5375.573,E2 -5375.573} C_VEL
LIN {X 0,Y 509.842,Z 198.606,A -85,B 0,C 180,E1 -5378.998,E2 -5378.998} C_VEL
LIN {X 0,Y 509.88,Z 198.59,A -85,B 0,C 180,E1 -5381.999,E2 -5381.999} C_VEL
LIN {X 0,Y 509.901,Z 198.597,A -85,B 0,C 180,E1 -5384.818,E2 -5384.818} C_VEL
LIN {X 0,Y 509.897,Z 198.591,A -85,B 0,C 180,E1 -5388.12,E2 -5388.12} C_VEL
LIN {X 0,Y 509.908,Z 198.591,A -85,B 0,C 180,E1 -5391.28,E2 -5391.28} C_VEL
LIN {X 0,Y 509.969,Z 198.58,A -85,B 0,C 180,E1 -5393.67,E2 -5393.67} C_VEL
LIN {X 0,Y 510.045,Z 198.572,A -85,B 0,C 180,E1 -5397.631,E2 -5397.631} C_VEL
LIN {X 0,Y 510.057,Z 198.578,A -85,B 0,C 180,E1 -5400.789,E2 -5400.789} C_VEL
LIN {X 0,Y 509.95,Z 198.583,A -85,B 0,C 180,E1 -5403.16,E2 -5403.16} C_VEL
LIN {X 0,Y 509.969,Z 198.587,A -85,B 0,C 180,E1 -5406.33,E2 -5406.33} C_VEL
LIN {X 0,Y 509.909,Z 198.594,A -85,B 0,C 180,E1 -5408.72,E2 -5408.72} C_VEL
LIN {X 0,Y 509.895,Z 198.593,A -85,B 0,C 180,E1 -5411.932,E2 -5411.932} C_VEL
LIN {X 0,Y 509.884,Z 198.594,A -85,B 0,C 180,E1 -5415.242,E2 -5415.242} C_VEL
LIN {X 0,Y 509.879,Z 198.593,A -85,B 0,C 180,E1 -5418.001,E2 -5418.001} C_VEL
LIN {X 0,Y 509.842,Z 198.597,A -85,B 0,C 180,E1 -5421.002,E2 -5421.002} C_VEL
LIN {X 0,Y 509.828,Z 198.601,A -85,B 0,C 180,E1 -5423.563,E2 -5423.563} C_VEL
LIN {X 0,Y 509.903,Z 198.597,A -85,B 0,C 180,E1 -5426.379,E2 -5426.379} C_VEL
LIN {X 0,Y 509.877,Z 198.595,A -85,B 0,C 180,E1 -5428.844,E2 -5428.844} C_VEL
LIN {X 0,Y 509.819,Z 198.602,A -85,B 0,C 180,E1 -5431.59,E2 -5431.59} C_VEL
LIN {X 0,Y 509.846,Z 198.602,A -85,B 0,C 180,E1 -5434.414,E2 -5434.414} C_VEL
LIN {X 0,Y 509.812,Z 198.601,A -85,B 0,C 180,E1 -5437.341,E2 -5437.341} C_VEL
LIN {X 0,Y 509.832,Z 198.596,A -85,B 0,C 180,E1 -5440.383,E2 -5440.383} C_VEL
LIN {X 0,Y 509.818,Z 198.601,A -85,B 0,C 180,E1 -5443.063,E2 -5443.063} C_VEL
LIN {X 0,Y 509.825,Z 198.606,A -85,B 0,C 180,E1 -5445.793,E2 -5445.793} C_VEL
LIN {X 0,Y 509.861,Z 198.597,A -85,B 0,C 180,E1 -5448.576,E2 -5448.576} C_VEL
LIN {X 0,Y 509.848,Z 198.602,A -85,B 0,C 180,E1 -5451.787,E2 -5451.787} C_VEL
LIN {X 0,Y 509.839,Z 198.6,A -85,B 0,C 180,E1 -5454.624,E2 -5454.624} C_VEL
LIN {X 0,Y 509.86,Z 198.601,A -85,B 0,C 180,E1 -5457.482,E2 -5457.482} C_VEL
LIN {X 0,Y 509.856,Z 198.603,A -85,B 0,C 180,E1 -5460.274,E2 -5460.274} C_VEL
LIN {X 0,Y 509.873,Z 198.602,A -85,B 0,C 180,E1 -5461.445,E2 -5461.445} C_VEL
LIN {X 0,Y 513.079,Z 212.434,A -85,B 0,C 180,E1 -5463.566,E2 -5463.566} C_VEL
LIN {X 0,Y 512.574,Z 229.761,A -85,B 0,C 180,E1 -5465.927,E2 -5465.927} C_VEL
LIN {X 0,Y 512.037,Z 244.433,A -85,B 0,C 180,E1 -5467.9,E2 -5467.9} C_VEL
LIN {X 0,Y 515.302,Z 261.598,A -85,B 0,C 180,E1 -5468.299,E2 -5468.299} C_VEL
LIN {X 0,Y 514.168,Z 410.043,A -85,B 0,C 180,E1 -5470.436,E2 -5470.436} C_VEL
LIN {X 0,Y 513.786,Z 425.612,A -85,B 0,C 180,E1 -5470.809,E2 -5470.809} C_VEL
LIN {X 0,Y 513.381,Z 440.605,A -85,B 0,C 180,E1 -5471.338,E2 -5471.338} C_VEL
LIN {X 0,Y 512.783,Z 455.626,A -85,B 0,C 180,E1 -5472.039,E2 -5472.039} C_VEL
LIN {X 0,Y 512.284,Z 469.143,A -85,B 0,C 180,E1 -5472.845,E2 -5472.845} C_VEL
LIN {X 0,Y 511.712,Z 481.607,A -85,B 0,C 180,E1 -5473.75,E2 -5473.75} C_VEL
LIN {X 0,Y 511.157,Z 494.287,A -85,B 0,C 180,E1 -5474.857,E2 -5474.857} C_VEL
LIN {X 0,Y 510.639,Z 505.808,A -85,B 0,C 180,E1 -5476.063,E2 -5476.063} C_VEL
LIN {X 0,Y 510.21,Z 515.508,A -85,B 0,C 180,E1 -5477.268,E2 -5477.268} C_VEL
LIN {X 0,Y 509.846,Z 525.192,A -85,B 0,C 180,E1 -5478.697,E2 -5478.697} C_VEL
LIN {X 0,Y 509.565,Z 532.975,A -85,B 0,C 180,E1 -5480.073,E2 -5480.073} C_VEL
LIN {X 0,Y 509.394,Z 540.389,A -85,B 0,C 180,E1 -5481.671,E2 -5481.671} C_VEL
LIN {X 0,Y 509.289,Z 546.271,A -85,B 0,C 180,E1 -5483.264,E2 -5483.264} C_VEL
LIN {X 0,Y 509.263,Z 549.766,A -85,B 0,C 180,E1 -5484.457,E2 -5484.457} C_VEL
LIN {X 0,Y 509.171,Z 553.298,A -85,B 0,C 180,E1 -5486.043,E2 -5486.043} C_VEL
LIN {X 0,Y 509.187,Z 555.622,A -85,B 0,C 180,E1 -5487.627,E2 -5487.627} C_VEL
LIN {X 0,Y 509.071,Z 556.789,A -85,B 0,C 180,E1 -5489.209,E2 -5489.209} C_VEL
LIN {X 0,Y 509.071,Z 556.788,A -85,B 0,C 180,E1 -5490.791,E2 -5490.791} C_VEL
LIN {X 0,Y 509.187,Z 555.618,A -85,B 0,C 180,E1 -5492.373,E2 -5492.373} C_VEL
LIN {X 0,Y 509.171,Z 553.293,A -85,B 0,C 180,E1 -5493.957,E2 -5493.957} C_VEL
LIN {X 0,Y 509.264,Z 549.768,A -85,B 0,C 180,E1 -5495.543,E2 -5495.543} C_VEL
LIN {X 0,Y 509.316,Z 544.948,A -85,B 0,C 180,E1 -5497.134,E2 -5497.134} C_VEL
LIN {X 0,Y 509.453,Z 538.706,A -85,B 0,C 180,E1 -5498.728,E2 -5498.728} C_VEL
LIN {X 0,Y 509.7,Z 530.868,A -85,B 0,C 180,E1 -5500.326,E2 -5500.326} C_VEL
LIN {X 0,Y 509.957,Z 522.391,A -85,B 0,C 180,E1 -5501.749,E2 -5501.749} C_VEL
LIN {X 0,Y 510.343,Z 512.493,A -85,B 0,C 180,E1 -5503.133,E2 -5503.133} C_VEL
LIN {X 0,Y 510.78,Z 502.225,A -85,B 0,C 180,E1 -5504.339,E2 -5504.339} C_VEL
LIN {X 0,Y 511.369,Z 489.426,A -85,B 0,C 180,E1 -5505.597,E2 -5505.597} C_VEL
LIN {X 0,Y 511.976,Z 476.39,A -85,B 0,C 180,E1 -5506.651,E2 -5506.651} C_VEL
LIN {X 0,Y 512.569,Z 462.749,A -85,B 0,C 180,E1 -5507.556,E2 -5507.556} C_VEL
LIN {X 0,Y 513.104,Z 448.626,A -85,B 0,C 180,E1 -5508.311,E2 -5508.311} C_VEL
LIN {X 0,Y 513.563,Z 434.138,A -85,B 0,C 180,E1 -5508.913,E2 -5508.913} C_VEL
LIN {X 0,Y 513.934,Z 418.679,A -85,B 0,C 180,E1 -5509.381,E2 -5509.381} C_VEL
LIN {X 0,Y 514.251,Z 402.339,A -85,B 0,C 180,E1 -5509.692,E2 -5509.692} C_VEL
LIN {X 0,Y 515.302,Z 261.597,A -85,B 0,C 180,E1 -5511.701,E2 -5511.701} C_VEL
LIN {X 0,Y 512.003,Z 244.408,A -85,B 0,C 180,E1 -5512.105,E2 -5512.105} C_VEL
LIN {X 0,Y 512.806,Z 223.461,A -85,B 0,C 180,E1 -5514.924,E2 -5514.924} C_VEL
LIN {X 0,Y 513.063,Z 212.429,A -85,B 0,C 180,E1 -5516.435,E2 -5516.435} C_VEL
LIN {X 0,Y 509.895,Z 198.598,A -85,B 0,C 180,E1 -5518.554,E2 -5518.554} C_VEL
LIN {X 0,Y 509.818,Z 198.601,A -85,B 0,C 180,E1 -5521.589,E2 -5521.589} C_VEL
LIN {X 0,Y 509.848,Z 198.6,A -85,B 0,C 180,E1 -5524.413,E2 -5524.413} C_VEL
LIN {X 0,Y 509.815,Z 198.602,A -85,B 0,C 180,E1 -5527.34,E2 -5527.34} C_VEL
LIN {X 0,Y 509.857,Z 198.6,A -85,B 0,C 180,E1 -5530.379,E2 -5530.379} C_VEL
LIN {X 0,Y 509.819,Z 198.6,A -85,B 0,C 180,E1 -5533.062,E2 -5533.062} C_VEL
LIN {X 0,Y 509.825,Z 198.604,A -85,B 0,C 180,E1 -5535.792,E2 -5535.792} C_VEL
LIN {X 0,Y 509.859,Z 198.595,A -85,B 0,C 180,E1 -5538.575,E2 -5538.575} C_VEL
LIN {X 0,Y 509.846,Z 198.602,A -85,B 0,C 180,E1 -5541.786,E2 -5541.786} C_VEL
LIN {X 0,Y 509.839,Z 198.596,A -85,B 0,C 180,E1 -5544.623,E2 -5544.623} C_VEL
LIN {X 0,Y 509.858,Z 198.597,A -85,B 0,C 180,E1 -5547.481,E2 -5547.481} C_VEL
LIN {X 0,Y 509.874,Z 198.594,A -85,B 0,C 180,E1 -5550.268,E2 -5550.268} C_VEL
LIN {X 0,Y 509.877,Z 198.592,A -85,B 0,C 180,E1 -5552.944,E2 -5552.944} C_VEL
LIN {X 0,Y 509.861,Z 198.602,A -85,B 0,C 180,E1 -5555.574,E2 -5555.574} C_VEL
LIN {X 0,Y 509.814,Z 198.595,A -85,B 0,C 180,E1 -5558.148,E2 -5558.148} C_VEL
LIN {X 0,Y 509.856,Z 198.594,A -85,B 0,C 180,E1 -5560.681,E2 -5560.681} C_VEL
LIN {X 0,Y 509.878,Z 198.595,A -85,B 0,C 180,E1 -5563.175,E2 -5563.175} C_VEL
LIN {X 0,Y 509.855,Z 198.603,A -85,B 0,C 180,E1 -5565.634,E2 -5565.634} C_VEL
LIN {X 0,Y 509.908,Z 198.589,A -85,B 0,C 180,E1 -5568.875,E2 -5568.875} C_VEL
LIN {X 0,Y 509.943,Z 198.585,A -85,B 0,C 180,E1 -5572.078,E2 -5572.078} C_VEL
LIN {X 0,Y 509.975,Z 198.58,A -85,B 0,C 180,E1 -5574.464,E2 -5574.464} C_VEL
LIN {X 0,Y 510.046,Z 198.578,A -85,B 0,C 180,E1 -5577.631,E2 -5577.631} C_VEL
LIN {X 0,Y 510.057,Z 198.57,A -85,B 0,C 180,E1 -5580.79,E2 -5580.79} C_VEL
LIN {X 0,Y 509.95,Z 198.59,A -85,B 0,C 180,E1 -5583.16,E2 -5583.16} C_VEL
LIN {X 0,Y 509.969,Z 198.582,A -85,B 0,C 180,E1 -5586.33,E2 -5586.33} C_VEL
LIN {X 0,Y 509.91,Z 198.589,A -85,B 0,C 180,E1 -5588.72,E2 -5588.72} C_VEL
LIN {X 0,Y 509.896,Z 198.59,A -85,B 0,C 180,E1 -5591.932,E2 -5591.932} C_VEL
LIN {X 0,Y 509.884,Z 198.599,A -85,B 0,C 180,E1 -5595.242,E2 -5595.242} C_VEL
LIN {X 0,Y 509.88,Z 198.593,A -85,B 0,C 180,E1 -5598.001,E2 -5598.001} C_VEL
LIN {X 0,Y 509.842,Z 198.603,A -85,B 0,C 180,E1 -5601.002,E2 -5601.002} C_VEL
LIN {X 0,Y 509.861,Z 198.595,A -85,B 0,C 180,E1 -5604.427,E2 -5604.427} C_VEL
LIN {X 0,Y 509.878,Z 198.593,A -85,B 0,C 180,E1 -5607.056,E2 -5607.056} C_VEL
LIN {X 0,Y 509.874,Z 198.594,A -85,B 0,C 180,E1 -5609.75,E2 -5609.75} C_VEL
LIN {X 0,Y 509.87,Z 198.6,A -85,B 0,C 180,E1 -5612.775,E2 -5612.775} C_VEL
LIN {X 0,Y 509.836,Z 198.598,A -85,B 0,C 180,E1 -5615.582,E2 -5615.582} C_VEL
LIN {X 0,Y 509.845,Z 198.598,A -85,B 0,C 180,E1 -5618.339,E2 -5618.339} C_VEL
LIN {X 0,Y 509.853,Z 198.595,A -85,B 0,C 180,E1 -5621.426,E2 -5621.426} C_VEL
LIN {X 0,Y 509.852,Z 198.602,A -85,B 0,C 180,E1 -5624.669,E2 -5624.669} C_VEL
LIN {X 0,Y 509.857,Z 198.597,A -85,B 0,C 180,E1 -5628.103,E2 -5628.103} C_VEL
LIN {X 0,Y 509.843,Z 198.602,A -85,B 0,C 180,E1 -5630.648,E2 -5630.648} C_VEL
LIN {X 0,Y 509.817,Z 198.6,A -85,B 0,C 180,E1 -5633.747,E2 -5633.747} C_VEL
LIN {X 0,Y 509.149,Z 198.688,A -85,B 0,C 180,E1 -5634.407,E2 -5634.407} C_VEL
LIN {X 0,Y 506.337,Z 199.039,A -85,B 0,C 180,E1 -5635.479,E2 -5635.479} C_VEL
LIN {X 0,Y 503.949,Z 199.338,A -85,B 0,C 180,E1 -5636.342,E2 -5636.342} C_VEL
LIN {X 0,Y 502.903,Z 199.467,A -85,B 0,C 180,E1 -5637.009,E2 -5637.009} C_VEL
LIN {X 0,Y 502.806,Z 199.477,A -85,B 0,C 180,E1 -5637.234,E2 -5637.234} C_VEL
LIN {X 0,Y 502.814,Z 199.478,A -85,B 0,C 180,E1 -5640.066,E2 -5640.066} C_VEL
LIN {X 0,Y 502.833,Z 199.477,A -85,B 0,C 180,E1 -5642.534,E2 -5642.534} C_VEL
LIN {X 0,Y 502.874,Z 199.673,A -85,B 0,C 180,E1 -5644.436,E2 -5644.436} C_VEL
LIN {X 0,Y 505.457,Z 211.955,A -85,B 0,C 180,E1 -5646.59,E2 -5646.59} C_VEL
LIN {X 0,Y 505.239,Z 218.58,A -85,B 0,C 180,E1 -5647.638,E2 -5647.638} C_VEL
LIN {X 0,Y 508.723,Z 233.753,A -85,B 0,C 180,E1 -5648.034,E2 -5648.034} C_VEL
LIN {X 0,Y 507.87,Z 350.651,A -85,B 0,C 180,E1 -5649.734,E2 -5649.734} C_VEL
LIN {X 0,Y 507.516,Z 384.834,A -85,B 0,C 180,E1 -5650.255,E2 -5650.255} C_VEL
LIN {X 0,Y 507.206,Z 400.219,A -85,B 0,C 180,E1 -5650.656,E2 -5650.656} C_VEL
LIN {X 0,Y 506.793,Z 414.678,A -85,B 0,C 180,E1 -5651.191,E2 -5651.191} C_VEL
LIN {X 0,Y 506.318,Z 427.36,A -85,B 0,C 180,E1 -5651.802,E2 -5651.802} C_VEL
LIN {X 0,Y 505.726,Z 440.957,A -85,B 0,C 180,E1 -5652.616,E2 -5652.616} C_VEL
LIN {X 0,Y 505.101,Z 453.589,A -85,B 0,C 180,E1 -5653.542,E2 -5653.542} C_VEL
LIN {X 0,Y 504.473,Z 466.108,A -85,B 0,C 180,E1 -5654.651,E2 -5654.651} C_VEL
LIN {X 0,Y 503.911,Z 477.574,A -85,B 0,C 180,E1 -5655.873,E2 -5655.873} C_VEL
LIN {X 0,Y 503.434,Z 487.222,A -85,B 0,C 180,E1 -5657.094,E2 -5657.094} C_VEL
LIN {X 0,Y 503.02,Z 496.844,A -85,B 0,C 180,E1 -5658.545,E2 -5658.545} C_VEL
LIN {X 0,Y 502.652,Z 505.544,A -85,B 0,C 180,E1 -5660.138,E2 -5660.138} C_VEL
LIN {X 0,Y 502.428,Z 511.889,A -85,B 0,C 180,E1 -5661.554,E2 -5661.554} C_VEL
LIN {X 0,Y 502.259,Z 517.842,A -85,B 0,C 180,E1 -5663.21,E2 -5663.21} C_VEL
LIN {X 0,Y 502.262,Z 521.168,A -85,B 0,C 180,E1 -5664.379,E2 -5664.379} C_VEL
LIN {X 0,Y 502.162,Z 524.669,A -85,B 0,C 180,E1 -5665.987,E2 -5665.987} C_VEL
LIN {X 0,Y 502.118,Z 526.987,A -85,B 0,C 180,E1 -5667.593,E2 -5667.593} C_VEL
LIN {X 0,Y 501.987,Z 528.177,A -85,B 0,C 180,E1 -5669.198,E2 -5669.198} C_VEL
LIN {X 0,Y 501.988,Z 528.196,A -85,B 0,C 180,E1 -5670.802,E2 -5670.802} C_VEL
LIN {X 0,Y 502.118,Z 527.08,A -85,B 0,C 180,E1 -5672.406,E2 -5672.406} C_VEL
LIN {X 0,Y 502.162,Z 524.835,A -85,B 0,C 180,E1 -5674.013,E2 -5674.013} C_VEL
LIN {X 0,Y 502.253,Z 521.403,A -85,B 0,C 180,E1 -5675.621,E2 -5675.621} C_VEL
LIN {X 0,Y 502.304,Z 516.705,A -85,B 0,C 180,E1 -5677.234,E2 -5677.234} C_VEL
LIN {X 0,Y 502.473,Z 510.616,A -85,B 0,C 180,E1 -5678.85,E2 -5678.85} C_VEL
LIN {X 0,Y 502.77,Z 502.945,A -85,B 0,C 180,E1 -5680.47,E2 -5680.47} C_VEL
LIN {X 0,Y 503.045,Z 494.79,A -85,B 0,C 180,E1 -5681.888,E2 -5681.888} C_VEL
LIN {X 0,Y 503.572,Z 484.911,A -85,B 0,C 180,E1 -5683.313,E2 -5683.313} C_VEL
LIN {X 0,Y 504.055,Z 474.805,A -85,B 0,C 180,E1 -5684.535,E2 -5684.535} C_VEL
LIN {X 0,Y 504.617,Z 463.544,A -85,B 0,C 180,E1 -5685.683,E2 -5685.683} C_VEL
LIN {X 0,Y 505.249,Z 450.706,A -85,B 0,C 180,E1 -5686.776,E2 -5686.776} C_VEL
LIN {X 0,Y 505.899,Z 437.594,A -85,B 0,C 180,E1 -5687.691,E2 -5687.691} C_VEL
LIN {X 0,Y 506.351,Z 425.11,A -85,B 0,C 180,E1 -5688.406,E2 -5688.406} C_VEL
LIN {X 0,Y 506.916,Z 410.622,A -85,B 0,C 180,E1 -5689.062,E2 -5689.062} C_VEL
LIN {X 0,Y 507.264,Z 395.631,A -85,B 0,C 180,E1 -5689.571,E2 -5689.571} C_VEL
LIN {X 0,Y 507.611,Z 379.511,A -85,B 0,C 180,E1 -5689.931,E2 -5689.931} C_VEL
LIN {X 0,Y 508.83,Z 234.747,A -85,B 0,C 180,E1 -5692.036,E2 -5692.036} C_VEL
LIN {X 0,Y 505.255,Z 218.537,A -85,B 0,C 180,E1 -5692.457,E2 -5692.457} C_VEL
LIN {X 0,Y 505.485,Z 211.786,A -85,B 0,C 180,E1 -5693.527,E2 -5693.527} C_VEL
LIN {X 0,Y 502.879,Z 199.473,A -85,B 0,C 180,E1 -5695.728,E2 -5695.728} C_VEL
LIN {X 0,Y 502.839,Z 199.474,A -85,B 0,C 180,E1 -5698.372,E2 -5698.372} C_VEL
LIN {X 0,Y 502.792,Z 199.484,A -85,B 0,C 180,E1 -5701.498,E2 -5701.498} C_VEL
LIN {X 0,Y 502.802,Z 199.476,A -85,B 0,C 180,E1 -5704.444,E2 -5704.444} C_VEL
LIN {X 0,Y 502.777,Z 199.482,A -85,B 0,C 180,E1 -5707.177,E2 -5707.177} C_VEL
LIN {X 0,Y 502.785,Z 199.477,A -85,B 0,C 180,E1 -5710.014,E2 -5710.014} C_VEL
LIN {X 0,Y 502.799,Z 199.475,A -85,B 0,C 180,E1 -5712.198,E2 -5712.198} C_VEL
LIN {X 0,Y 502.796,Z 199.481,A -85,B 0,C 180,E1 -5715.467,E2 -5715.467} C_VEL
LIN {X 0,Y 502.821,Z 199.474,A -85,B 0,C 180,E1 -5719.003,E2 -5719.003} C_VEL
LIN {X 0,Y 502.788,Z 199.47,A -85,B 0,C 180,E1 -5722.045,E2 -5722.045} C_VEL
LIN {X 0,Y 502.803,Z 199.48,A -85,B 0,C 180,E1 -5725.034,E2 -5725.034} C_VEL
LIN {X 0,Y 502.781,Z 199.47,A -85,B 0,C 180,E1 -5727.915,E2 -5727.915} C_VEL
LIN {X 0,Y 502.832,Z 199.471,A -85,B 0,C 180,E1 -5730.713,E2 -5730.713} C_VEL
LIN {X 0,Y 502.855,Z 199.469,A -85,B 0,C 180,E1 -5733.439,E2 -5733.439} C_VEL
LIN {X 0,Y 502.783,Z 199.477,A -85,B 0,C 180,E1 -5736.086,E2 -5736.086} C_VEL
LIN {X 0,Y 502.775,Z 199.481,A -85,B 0,C 180,E1 -5738.688,E2 -5738.688} C_VEL
LIN {X 0,Y 502.822,Z 199.474,A -85,B 0,C 180,E1 -5741.248,E2 -5741.248} C_VEL
LIN {X 0,Y 502.815,Z 199.473,A -85,B 0,C 180,E1 -5743.767,E2 -5743.767} C_VEL
LIN {X 0,Y 502.826,Z 199.469,A -85,B 0,C 180,E1 -5746.254,E2 -5746.254} C_VEL
LIN {X 0,Y 502.872,Z 199.473,A -85,B 0,C 180,E1 -5748.717,E2 -5748.717} C_VEL
LIN {X 0,Y 502.892,Z 199.463,A -85,B 0,C 180,E1 -5751.966,E2 -5751.966} C_VEL
LIN {X 0,Y 502.93,Z 199.461,A -85,B 0,C 180,E1 -5754.386,E2 -5754.386} C_VEL
LIN {X 0,Y 503.015,Z 199.448,A -85,B 0,C 180,E1 -5757.598,E2 -5757.598} C_VEL
LIN {X 0,Y 503.016,Z 199.445,A -85,B 0,C 180,E1 -5760,E2 -5760} C_VEL
LIN {X 0,Y 503.015,Z 199.453,A -85,B 0,C 180,E1 -5762.402,E2 -5762.402} C_VEL
LIN {X 0,Y 502.93,Z 199.458,A -85,B 0,C 180,E1 -5765.613,E2 -5765.613} C_VEL
LIN {X 0,Y 502.893,Z 199.464,A -85,B 0,C 180,E1 -5768.033,E2 -5768.033} C_VEL
LIN {X 0,Y 502.872,Z 199.467,A -85,B 0,C 180,E1 -5771.283,E2 -5771.283} C_VEL
LIN {X 0,Y 502.842,Z 199.478,A -85,B 0,C 180,E1 -5774.571,E2 -5774.571} C_VEL
LIN {X 0,Y 502.853,Z 199.468,A -85,B 0,C 180,E1 -5777.907,E2 -5777.907} C_VEL
LIN {X 0,Y 502.819,Z 199.477,A -85,B 0,C 180,E1 -5780.536,E2 -5780.536} C_VEL
LIN {X 0,Y 502.788,Z 199.478,A -85,B 0,C 180,E1 -5783.041,E2 -5783.041} C_VEL
LIN {X 0,Y 502.831,Z 199.47,A -85,B 0,C 180,E1 -5785.676,E2 -5785.676} C_VEL
LIN {X 0,Y 502.834,Z 199.478,A -85,B 0,C 180,E1 -5788.373,E2 -5788.373} C_VEL
LIN {X 0,Y 502.789,Z 199.477,A -85,B 0,C 180,E1 -5791.5,E2 -5791.5} C_VEL
LIN {X 0,Y 502.799,Z 199.48,A -85,B 0,C 180,E1 -5794.445,E2 -5794.445} C_VEL
LIN {X 0,Y 502.774,Z 199.478,A -85,B 0,C 180,E1 -5797.179,E2 -5797.179} C_VEL
LIN {X 0,Y 502.781,Z 199.476,A -85,B 0,C 180,E1 -5800.016,E2 -5800.016} C_VEL
LIN {X 0,Y 502.796,Z 199.481,A -85,B 0,C 180,E1 -5802.2,E2 -5802.2} C_VEL
LIN {X 0,Y 502.795,Z 199.478,A -85,B 0,C 180,E1 -5805.469,E2 -5805.469} C_VEL
LIN {X 0,Y 502.822,Z 199.472,A -85,B 0,C 180,E1 -5809.005,E2 -5809.005} C_VEL
LIN {X 0,Y 502.79,Z 199.478,A -85,B 0,C 180,E1 -5812.047,E2 -5812.047} C_VEL
LIN {X 0,Y 502.804,Z 199.476,A -85,B 0,C 180,E1 -5815.035,E2 -5815.035} C_VEL
LIN {X 0,Y 502.781,Z 199.485,A -85,B 0,C 180,E1 -5817.916,E2 -5817.916} C_VEL
LIN {X 0,Y 502.865,Z 199.548,A -85,B 0,C 180,E1 -5821.174,E2 -5821.174} C_VEL
LIN {X 0,Y 506.256,Z 214.074,A -85,B 0,C 180,E1 -5823.44,E2 -5823.44} C_VEL
LIN {X 0,Y 505.704,Z 231.14,A -85,B 0,C 180,E1 -5825.797,E2 -5825.797} C_VEL
LIN {X 0,Y 505.187,Z 244.159,A -85,B 0,C 180,E1 -5827.574,E2 -5827.574} C_VEL
LIN {X 0,Y 508.706,Z 262.427,A -85,B 0,C 180,E1 -5828.018,E2 -5828.018} C_VEL
LIN {X 0,Y 507.471,Z 410.54,A -85,B 0,C 180,E1 -5830.179,E2 -5830.179} C_VEL
LIN {X 0,Y 507.039,Z 426.276,A -85,B 0,C 180,E1 -5830.57,E2 -5830.57} C_VEL
LIN {X 0,Y 506.572,Z 441.863,A -85,B 0,C 180,E1 -5831.14,E2 -5831.14} C_VEL
LIN {X 0,Y 506.005,Z 455.424,A -85,B 0,C 180,E1 -5831.79,E2 -5831.79} C_VEL
LIN {X 0,Y 505.47,Z 468.941,A -85,B 0,C 180,E1 -5832.607,E2 -5832.607} C_VEL
LIN {X 0,Y 504.82,Z 481.403,A -85,B 0,C 180,E1 -5833.522,E2 -5833.522} C_VEL
LIN {X 0,Y 504.247,Z 494.084,A -85,B 0,C 180,E1 -5834.644,E2 -5834.644} C_VEL
LIN {X 0,Y 503.667,Z 505.605,A -85,B 0,C 180,E1 -5835.866,E2 -5835.866} C_VEL
LIN {X 0,Y 503.19,Z 515.304,A -85,B 0,C 180,E1 -5837.087,E2 -5837.087} C_VEL
LIN {X 0,Y 502.804,Z 525,A -85,B 0,C 180,E1 -5838.539,E2 -5838.539} C_VEL
LIN {X 0,Y 502.524,Z 532.773,A -85,B 0,C 180,E1 -5839.932,E2 -5839.932} C_VEL
LIN {X 0,Y 502.323,Z 540.187,A -85,B 0,C 180,E1 -5841.553,E2 -5841.553} C_VEL
LIN {X 0,Y 502.222,Z 546.07,A -85,B 0,C 180,E1 -5843.169,E2 -5843.169} C_VEL
LIN {X 0,Y 502.175,Z 549.565,A -85,B 0,C 180,E1 -5844.378,E2 -5844.378} C_VEL
LIN {X 0,Y 502.068,Z 553.096,A -85,B 0,C 180,E1 -5845.987,E2 -5845.987} C_VEL
LIN {X 0,Y 502.088,Z 555.421,A -85,B 0,C 180,E1 -5847.593,E2 -5847.593} C_VEL
LIN {X 0,Y 501.988,Z 556.589,A -85,B 0,C 180,E1 -5849.198,E2 -5849.198} C_VEL
LIN {X 0,Y 501.988,Z 556.588,A -85,B 0,C 180,E1 -5850.802,E2 -5850.802} C_VEL
LIN {X 0,Y 502.088,Z 555.417,A -85,B 0,C 180,E1 -5852.407,E2 -5852.407} C_VEL
LIN {X 0,Y 502.068,Z 553.091,A -85,B 0,C 180,E1 -5854.013,E2 -5854.013} C_VEL
LIN {X 0,Y 502.177,Z 549.566,A -85,B 0,C 180,E1 -5855.622,E2 -5855.622} C_VEL
LIN {X 0,Y 502.24,Z 544.746,A -85,B 0,C 180,E1 -5857.235,E2 -5857.235} C_VEL
LIN {X 0,Y 502.363,Z 538.503,A -85,B 0,C 180,E1 -5858.852,E2 -5858.852} C_VEL
LIN {X 0,Y 502.635,Z 530.665,A -85,B 0,C 180,E1 -5860.473,E2 -5860.473} C_VEL
LIN {X 0,Y 502.869,Z 521.924,A -85,B 0,C 180,E1 -5861.957,E2 -5861.957} C_VEL
LIN {X 0,Y 503.353,Z 512.289,A -85,B 0,C 180,E1 -5863.319,E2 -5863.319} C_VEL
LIN {X 0,Y 503.823,Z 502.021,A -85,B 0,C 180,E1 -5864.542,E2 -5864.542} C_VEL
LIN {X 0,Y 504.439,Z 489.822,A -85,B 0,C 180,E1 -5865.761,E2 -5865.761} C_VEL
LIN {X 0,Y 505.089,Z 476.186,A -85,B 0,C 180,E1 -5866.885,E2 -5866.885} C_VEL
LIN {X 0,Y 505.75,Z 462.547,A -85,B 0,C 180,E1 -5867.801,E2 -5867.801} C_VEL
LIN {X 0,Y 506.329,Z 448.424,A -85,B 0,C 180,E1 -5868.565,E2 -5868.565} C_VEL
LIN {X 0,Y 506.855,Z 433.267,A -85,B 0,C 180,E1 -5869.197,E2 -5869.197} C_VEL
LIN {X 0,Y 507.282,Z 418.018,A -85,B 0,C 180,E1 -5869.657,E2 -5869.657} C_VEL
LIN {X 0,Y 507.554,Z 402.137,A -85,B 0,C 180,E1 -5869.962,E2 -5869.962} C_VEL
LIN {X 0,Y 508.712,Z 262.762,A -85,B 0,C 180,E1 -5871.977,E2 -5871.977} C_VEL
LIN {X 0,Y 505.187,Z 244.206,A -85,B 0,C 180,E1 -5872.419,E2 -5872.419} C_VEL
LIN {X 0,Y 506.084,Z 221.696,A -85,B 0,C 180,E1 -5875.498,E2 -5875.498} C_VEL
LIN {X 0,Y 506.22,Z 214.079,A -85,B 0,C 180,E1 -5876.561,E2 -5876.561} C_VEL
LIN {X 0,Y 502.844,Z 199.474,A -85,B 0,C 180,E1 -5878.856,E2 -5878.856} C_VEL
LIN {X 0,Y 502.782,Z 199.48,A -85,B 0,C 180,E1 -5882.084,E2 -5882.084} C_VEL
LIN {X 0,Y 502.804,Z 199.473,A -85,B 0,C 180,E1 -5884.965,E2 -5884.965} C_VEL
LIN {X 0,Y 502.79,Z 199.483,A -85,B 0,C 180,E1 -5887.953,E2 -5887.953} C_VEL
LIN {X 0,Y 502.822,Z 199.472,A -85,B 0,C 180,E1 -5891.065,E2 -5891.065} C_VEL
LIN {X 0,Y 502.795,Z 199.476,A -85,B 0,C 180,E1 -5894.531,E2 -5894.531} C_VEL
LIN {X 0,Y 502.794,Z 199.481,A -85,B 0,C 180,E1 -5897.861,E2 -5897.861} C_VEL
LIN {X 0,Y 502.814,Z 199.476,A -85,B 0,C 180,E1 -5900.24,E2 -5900.24} C_VEL
LIN {X 0,Y 502.771,Z 199.477,A -85,B 0,C 180,E1 -5903.053,E2 -5903.053} C_VEL
LIN {X 0,Y 502.801,Z 199.478,A -85,B 0,C 180,E1 -5906.006,E2 -5906.006} C_VEL
LIN {X 0,Y 502.792,Z 199.475,A -85,B 0,C 180,E1 -5908.857,E2 -5908.857} C_VEL
LIN {X 0,Y 502.837,Z 199.477,A -85,B 0,C 180,E1 -5911.704,E2 -5911.704} C_VEL
LIN {X 0,Y 502.832,Z 199.472,A -85,B 0,C 180,E1 -5914.324,E2 -5914.324} C_VEL
LIN {X 0,Y 502.79,Z 199.476,A -85,B 0,C 180,E1 -5917.298,E2 -5917.298} C_VEL
LIN {X 0,Y 502.817,Z 199.472,A -85,B 0,C 180,E1 -5920.4,E2 -5920.4} C_VEL
LIN {X 0,Y 502.827,Z 199.472,A -85,B 0,C 180,E1 -5922.932,E2 -5922.932} C_VEL
LIN {X 0,Y 502.836,Z 199.476,A -85,B 0,C 180,E1 -5925.429,E2 -5925.429} C_VEL
LIN {X 0,Y 502.872,Z 199.465,A -85,B 0,C 180,E1 -5928.717,E2 -5928.717} C_VEL
LIN {X 0,Y 502.893,Z 199.464,A -85,B 0,C 180,E1 -5931.967,E2 -5931.967} C_VEL
LIN {X 0,Y 502.931,Z 199.458,A -85,B 0,C 180,E1 -5934.387,E2 -5934.387} C_VEL
LIN {X 0,Y 503.015,Z 199.454,A -85,B 0,C 180,E1 -5937.598,E2 -5937.598} C_VEL
LIN {X 0,Y 503.016,Z 199.446,A -85,B 0,C 180,E1 -5940,E2 -5940} C_VEL
LIN {X 0,Y 503.015,Z 199.448,A -85,B 0,C 180,E1 -5942.402,E2 -5942.402} C_VEL
LIN {X 0,Y 502.939,Z 199.462,A -85,B 0,C 180,E1 -5945.614,E2 -5945.614} C_VEL
LIN {X 0,Y 502.893,Z 199.461,A -85,B 0,C 180,E1 -5948.034,E2 -5948.034} C_VEL
LIN {X 0,Y 502.872,Z 199.472,A -85,B 0,C 180,E1 -5951.283,E2 -5951.283} C_VEL
LIN {X 0,Y 502.836,Z 199.471,A -85,B 0,C 180,E1 -5954.571,E2 -5954.571} C_VEL
LIN {X 0,Y 502.853,Z 199.468,A -85,B 0,C 180,E1 -5957.907,E2 -5957.907} C_VEL
LIN {X 0,Y 502.82,Z 199.473,A -85,B 0,C 180,E1 -5960.537,E2 -5960.537} C_VEL
LIN {X 0,Y 502.786,Z 199.484,A -85,B 0,C 180,E1 -5963.041,E2 -5963.041} C_VEL
LIN {X 0,Y 502.832,Z 199.461,A -85,B 0,C 180,E1 -5965.676,E2 -5965.676} C_VEL
LIN {X 0,Y 502.835,Z 199.47,A -85,B 0,C 180,E1 -5968.373,E2 -5968.373} C_VEL
LIN {X 0,Y 502.79,Z 199.478,A -85,B 0,C 180,E1 -5971.5,E2 -5971.5} C_VEL
LIN {X 0,Y 502.8,Z 199.475,A -85,B 0,C 180,E1 -5974.445,E2 -5974.445} C_VEL
LIN {X 0,Y 502.775,Z 199.482,A -85,B 0,C 180,E1 -5977.179,E2 -5977.179} C_VEL
LIN {X 0,Y 502.783,Z 199.475,A -85,B 0,C 180,E1 -5980.016,E2 -5980.016} C_VEL
LIN {X 0,Y 502.798,Z 199.474,A -85,B 0,C 180,E1 -5982.2,E2 -5982.2} C_VEL
LIN {X 0,Y 502.796,Z 199.476,A -85,B 0,C 180,E1 -5985.469,E2 -5985.469} C_VEL
LIN {X 0,Y 502.826,Z 199.472,A -85,B 0,C 180,E1 -5987.865,E2 -5987.865} C_VEL
LIN {X 0,Y 502.798,Z 199.478,A -85,B 0,C 180,E1 -5991.025,E2 -5991.025} C_VEL
LIN {X 0,Y 502.772,Z 199.481,A -85,B 0,C 180,E1 -5994.17,E2 -5994.17} C_VEL
LIN {X 0,Y 502.806,Z 199.477,A -85,B 0,C 180,E1 -5997.234,E2 -5997.234} C_VEL
LIN {X 0,Y 502.105,Z 199.565,A -85,B 0,C 180,E1 -5997.903,E2 -5997.903} C_VEL
LIN {X 0,Y 499.241,Z 199.923,A -85,B 0,C 180,E1 -5998.989,E2 -5998.989} C_VEL
LIN {X 0,Y 496.846,Z 200.222,A -85,B 0,C 180,E1 -5999.864,E2 -5999.864} C_VEL
LIN {X 0,Y 495.83,Z 200.349,A -85,B 0,C 180,E1 -6000.539,E2 -6000.539} C_VEL
LIN {X 0,Y 495.752,Z 200.357,A -85,B 0,C 180,E1 -6000.768,E2 -6000.768} C_VEL
LIN {X 0,Y 495.819,Z 200.352,A -85,B 0,C 180,E1 -6004.047,E2 -6004.047} C_VEL
LIN {X 0,Y 495.842,Z 200.535,A -85,B 0,C 180,E1 -6004.161,E2 -6004.161} C_VEL
LIN {X 0,Y 498.566,Z 213.008,A -85,B 0,C 180,E1 -6006.387,E2 -6006.387} C_VEL
LIN {X 0,Y 498.448,Z 218.778,A -85,B 0,C 180,E1 -6007.316,E2 -6007.316} C_VEL
LIN {X 0,Y 502.172,Z 234.838,A -85,B 0,C 180,E1 -6007.746,E2 -6007.746} C_VEL
LIN {X 0,Y 501.243,Z 350.885,A -85,B 0,C 180,E1 -6009.454,E2 -6009.454} C_VEL
LIN {X 0,Y 500.84,Z 385.157,A -85,B 0,C 180,E1 -6009.983,E2 -6009.983} C_VEL
LIN {X 0,Y 500.532,Z 400.435,A -85,B 0,C 180,E1 -6010.387,E2 -6010.387} C_VEL
LIN {X 0,Y 500.08,Z 414.89,A -85,B 0,C 180,E1 -6010.929,E2 -6010.929} C_VEL
LIN {X 0,Y 499.571,Z 427.571,A -85,B 0,C 180,E1 -6011.547,E2 -6011.547} C_VEL
LIN {X 0,Y 498.942,Z 441.167,A -85,B 0,C 180,E1 -6012.372,E2 -6012.372} C_VEL
LIN {X 0,Y 498.23,Z 454.951,A -85,B 0,C 180,E1 -6013.403,E2 -6013.403} C_VEL
LIN {X 0,Y 497.556,Z 467.379,A -85,B 0,C 180,E1 -6014.538,E2 -6014.538} C_VEL
LIN {X 0,Y 497.001,Z 477.782,A -85,B 0,C 180,E1 -6015.673,E2 -6015.673} C_VEL
LIN {X 0,Y 496.481,Z 487.428,A -85,B 0,C 180,E1 -6016.91,E2 -6016.91} C_VEL
LIN {X 0,Y 496.044,Z 496.455,A -85,B 0,C 180,E1 -6018.28,E2 -6018.28} C_VEL
LIN {X 0,Y 495.658,Z 504.749,A -85,B 0,C 180,E1 -6019.791,E2 -6019.791} C_VEL
LIN {X 0,Y 495.374,Z 512.094,A -85,B 0,C 180,E1 -6021.433,E2 -6021.433} C_VEL
LIN {X 0,Y 495.198,Z 517.922,A -85,B 0,C 180,E1 -6023.071,E2 -6023.071} C_VEL
LIN {X 0,Y 495.199,Z 521.37,A -85,B 0,C 180,E1 -6024.299,E2 -6024.299} C_VEL
LIN {X 0,Y 495.061,Z 524.872,A -85,B 0,C 180,E1 -6025.93,E2 -6025.93} C_VEL
LIN {X 0,Y 495.021,Z 527.189,A -85,B 0,C 180,E1 -6027.559,E2 -6027.559} C_VEL
LIN {X 0,Y 494.907,Z 528.378,A -85,B 0,C 180,E1 -6029.186,E2 -6029.186} C_VEL
LIN {X 0,Y 494.908,Z 528.396,A -85,B 0,C 180,E1 -6030.814,E2 -6030.814} C_VEL
LIN {X 0,Y 495.022,Z 527.28,A -85,B 0,C 180,E1 -6032.441,E2 -6032.441} C_VEL
LIN {X 0,Y 495.061,Z 525.035,A -85,B 0,C 180,E1 -6034.07,E2 -6034.07} C_VEL
LIN {X 0,Y 495.189,Z 521.602,A -85,B 0,C 180,E1 -6035.701,E2 -6035.701} C_VEL
LIN {X 0,Y 495.242,Z 516.904,A -85,B 0,C 180,E1 -6037.338,E2 -6037.338} C_VEL
LIN {X 0,Y 495.44,Z 510.814,A -85,B 0,C 180,E1 -6038.977,E2 -6038.977} C_VEL
LIN {X 0,Y 495.763,Z 503.143,A -85,B 0,C 180,E1 -6040.619,E2 -6040.619} C_VEL
LIN {X 0,Y 496.119,Z 494.135,A -85,B 0,C 180,E1 -6042.19,E2 -6042.19} C_VEL
LIN {X 0,Y 496.638,Z 485.108,A -85,B 0,C 180,E1 -6043.503,E2 -6043.503} C_VEL
LIN {X 0,Y 497.154,Z 475.001,A -85,B 0,C 180,E1 -6044.741,E2 -6044.741} C_VEL
LIN {X 0,Y 497.742,Z 464.019,A -85,B 0,C 180,E1 -6045.878,E2 -6045.878} C_VEL
LIN {X 0,Y 498.384,Z 452.184,A -85,B 0,C 180,E1 -6046.908,E2 -6046.908} C_VEL
LIN {X 0,Y 499.037,Z 439.362,A -85,B 0,C 180,E1 -6047.836,E2 -6047.836} C_VEL
LIN {X 0,Y 499.622,Z 425.3,A -85,B 0,C 180,E1 -6048.663,E2 -6048.663} C_VEL
LIN {X 0,Y 500.247,Z 410.007,A -85,B 0,C 180,E1 -6049.359,E2 -6049.359} C_VEL
LIN {X 0,Y 500.634,Z 395.36,A -85,B 0,C 180,E1 -6049.854,E2 -6049.854} C_VEL
LIN {X 0,Y 500.94,Z 381.054,A -85,B 0,C 180,E1 -6050.183,E2 -6050.183} C_VEL
LIN {X 0,Y 502.211,Z 235.267,A -85,B 0,C 180,E1 -6052.337,E2 -6052.337} C_VEL
LIN {X 0,Y 498.465,Z 218.752,A -85,B 0,C 180,E1 -6052.777,E2 -6052.777} C_VEL
LIN {X 0,Y 498.622,Z 213.457,A -85,B 0,C 180,E1 -6053.628,E2 -6053.628} C_VEL
LIN {X 0,Y 495.835,Z 200.349,A -85,B 0,C 180,E1 -6055.98,E2 -6055.98} C_VEL
LIN {X 0,Y 495.771,Z 200.354,A -85,B 0,C 180,E1 -6058.814,E2 -6058.814} C_VEL
LIN {X 0,Y 495.755,Z 200.36,A -85,B 0,C 180,E1 -6061.725,E2 -6061.725} C_VEL
LIN {X 0,Y 495.772,Z 200.353,A -85,B 0,C 180,E1 -6064.694,E2 -6064.694} C_VEL
LIN {X 0,Y 495.729,Z 200.365,A -85,B 0,C 180,E1 -6067.561,E2 -6067.561} C_VEL
LIN {X 0,Y 495.763,Z 200.352,A -85,B 0,C 180,E1 -6070.699,E2 -6070.699} C_VEL
LIN {X 0,Y 495.731,Z 200.359,A -85,B 0,C 180,E1 -6073.695,E2 -6073.695} C_VEL
LIN {X 0,Y 495.724,Z 200.356,A -85,B 0,C 180,E1 -6076.305,E2 -6076.305} C_VEL
LIN {X 0,Y 495.773,Z 200.357,A -85,B 0,C 180,E1 -6079.301,E2 -6079.301} C_VEL
LIN {X 0,Y 495.725,Z 200.35,A -85,B 0,C 180,E1 -6082.438,E2 -6082.438} C_VEL
LIN {X 0,Y 495.779,Z 200.354,A -85,B 0,C 180,E1 -6085.457,E2 -6085.457} C_VEL
LIN {X 0,Y 495.752,Z 200.345,A -85,B 0,C 180,E1 -6088.363,E2 -6088.363} C_VEL
LIN {X 0,Y 495.783,Z 200.352,A -85,B 0,C 180,E1 -6091.506,E2 -6091.506} C_VEL
LIN {X 0,Y 495.783,Z 200.347,A -85,B 0,C 180,E1 -6093.932,E2 -6093.932} C_VEL
LIN {X 0,Y 495.753,Z 200.356,A -85,B 0,C 180,E1 -6097.138,E2 -6097.138} C_VEL
LIN {X 0,Y 495.77,Z 200.351,A -85,B 0,C 180,E1 -6100.109,E2 -6100.109} C_VEL
LIN {X 0,Y 495.78,Z 200.352,A -85,B 0,C 180,E1 -6102.681,E2 -6102.681} C_VEL
LIN {X 0,Y 495.781,Z 200.349,A -85,B 0,C 180,E1 -6105.217,E2 -6105.217} C_VEL
LIN {X 0,Y 495.846,Z 200.346,A -85,B 0,C 180,E1 -6108.555,E2 -6108.555} C_VEL
LIN {X 0,Y 495.864,Z 200.338,A -85,B 0,C 180,E1 -6111.852,E2 -6111.852} C_VEL
LIN {X 0,Y 495.888,Z 200.337,A -85,B 0,C 180,E1 -6114.306,E2 -6114.306} C_VEL
LIN {X 0,Y 495.984,Z 200.324,A -85,B 0,C 180,E1 -6117.564,E2 -6117.564} C_VEL
LIN {X 0,Y 495.987,Z 200.321,A -85,B 0,C 180,E1 -6120,E2 -6120} C_VEL
LIN {X 0,Y 495.984,Z 200.33,A -85,B 0,C 180,E1 -6122.436,E2 -6122.436} C_VEL
LIN {X 0,Y 495.888,Z 200.336,A -85,B 0,C 180,E1 -6125.693,E2 -6125.693} C_VEL
LIN {X 0,Y 495.864,Z 200.341,A -85,B 0,C 180,E1 -6128.148,E2 -6128.148} C_VEL
LIN {X 0,Y 495.845,Z 200.341,A -85,B 0,C 180,E1 -6131.445,E2 -6131.445} C_VEL
LIN {X 0,Y 495.785,Z 200.354,A -85,B 0,C 180,E1 -6134.783,E2 -6134.783} C_VEL
LIN {X 0,Y 495.779,Z 200.346,A -85,B 0,C 180,E1 -6137.319,E2 -6137.319} C_VEL
LIN {X 0,Y 495.769,Z 200.354,A -85,B 0,C 180,E1 -6139.89,E2 -6139.89} C_VEL
LIN {X 0,Y 495.749,Z 200.356,A -85,B 0,C 180,E1 -6142.861,E2 -6142.861} C_VEL
LIN {X 0,Y 495.782,Z 200.352,A -85,B 0,C 180,E1 -6146.068,E2 -6146.068} C_VEL
LIN {X 0,Y 495.772,Z 200.353,A -85,B 0,C 180,E1 -6148.815,E2 -6148.815} C_VEL
LIN {X 0,Y 495.751,Z 200.356,A -85,B 0,C 180,E1 -6151.727,E2 -6151.727} C_VEL
LIN {X 0,Y 495.769,Z 200.353,A -85,B 0,C 180,E1 -6154.696,E2 -6154.696} C_VEL
LIN {X 0,Y 495.724,Z 200.358,A -85,B 0,C 180,E1 -6157.562,E2 -6157.562} C_VEL
LIN {X 0,Y 495.76,Z 200.347,A -85,B 0,C 180,E1 -6160.7,E2 -6160.7} C_VEL
LIN {X 0,Y 495.728,Z 200.362,A -85,B 0,C 180,E1 -6164.002,E2 -6164.002} C_VEL
LIN {X 0,Y 495.721,Z 200.357,A -85,B 0,C 180,E1 -6167.118,E2 -6167.118} C_VEL
LIN {X 0,Y 495.785,Z 200.354,A -85,B 0,C 180,E1 -6169.949,E2 -6169.949} C_VEL
LIN {X 0,Y 495.726,Z 200.356,A -85,B 0,C 180,E1 -6172.553,E2 -6172.553} C_VEL
LIN {X 0,Y 495.78,Z 200.354,A -85,B 0,C 180,E1 -6175.458,E2 -6175.458} C_VEL
LIN {X 0,Y 495.753,Z 200.356,A -85,B 0,C 180,E1 -6178.364,E2 -6178.364} C_VEL
LIN {X 0,Y 495.807,Z 200.538,A -85,B 0,C 180,E1 -6180.898,E2 -6180.898} C_VEL
LIN {X 0,Y 499.286,Z 215.208,A -85,B 0,C 180,E1 -6183.229,E2 -6183.229} C_VEL
LIN {X 0,Y 499.47,Z 218.364,A -85,B 0,C 180,E1 -6183.69,E2 -6183.69} C_VEL
LIN {X 0,Y 498.517,Z 240.355,A -85,B 0,C 180,E1 -6186.751,E2 -6186.751} C_VEL
LIN {X 0,Y 498.347,Z 243.958,A -85,B 0,C 180,E1 -6187.249,E2 -6187.249} C_VEL
LIN {X 0,Y 502.051,Z 262.932,A -85,B 0,C 180,E1 -6187.722,E2 -6187.722} C_VEL
LIN {X 0,Y 500.847,Z 403.75,A -85,B 0,C 180,E1 -6189.788,E2 -6189.788} C_VEL
LIN {X 0,Y 500.562,Z 419.284,A -85,B 0,C 180,E1 -6190.109,E2 -6190.109} C_VEL
LIN {X 0,Y 500.11,Z 434.053,A -85,B 0,C 180,E1 -6190.572,E2 -6190.572} C_VEL
LIN {X 0,Y 499.5,Z 449.245,A -85,B 0,C 180,E1 -6191.225,E2 -6191.225} C_VEL
LIN {X 0,Y 498.919,Z 462.353,A -85,B 0,C 180,E1 -6191.947,E2 -6191.947} C_VEL
LIN {X 0,Y 498.247,Z 475.978,A -85,B 0,C 180,E1 -6192.876,E2 -6192.876} C_VEL
LIN {X 0,Y 497.553,Z 489.292,A -85,B 0,C 180,E1 -6193.985,E2 -6193.985} C_VEL
LIN {X 0,Y 496.853,Z 501.816,A -85,B 0,C 180,E1 -6195.25,E2 -6195.25} C_VEL
LIN {X 0,Y 496.386,Z 512.086,A -85,B 0,C 180,E1 -6196.49,E2 -6196.49} C_VEL
LIN {X 0,Y 495.878,Z 522.159,A -85,B 0,C 180,E1 -6197.939,E2 -6197.939} C_VEL
LIN {X 0,Y 495.596,Z 530.469,A -85,B 0,C 180,E1 -6199.377,E2 -6199.377} C_VEL
LIN {X 0,Y 495.287,Z 538.304,A -85,B 0,C 180,E1 -6201.02,E2 -6201.02} C_VEL
LIN {X 0,Y 495.158,Z 544.54,A -85,B 0,C 180,E1 -6202.661,E2 -6202.661} C_VEL
LIN {X 0,Y 495.07,Z 549.363,A -85,B 0,C 180,E1 -6204.297,E2 -6204.297} C_VEL
LIN {X 0,Y 494.967,Z 552.895,A -85,B 0,C 180,E1 -6205.929,E2 -6205.929} C_VEL
LIN {X 0,Y 494.994,Z 555.221,A -85,B 0,C 180,E1 -6207.559,E2 -6207.559} C_VEL
LIN {X 0,Y 494.908,Z 556.388,A -85,B 0,C 180,E1 -6209.186,E2 -6209.186} C_VEL
LIN {X 0,Y 494.908,Z 556.387,A -85,B 0,C 180,E1 -6210.814,E2 -6210.814} C_VEL
LIN {X 0,Y 494.994,Z 555.216,A -85,B 0,C 180,E1 -6212.441,E2 -6212.441} C_VEL
LIN {X 0,Y 494.967,Z 552.89,A -85,B 0,C 180,E1 -6214.071,E2 -6214.071} C_VEL
LIN {X 0,Y 495.074,Z 549.364,A -85,B 0,C 180,E1 -6215.703,E2 -6215.703} C_VEL
LIN {X 0,Y 495.159,Z 544.544,A -85,B 0,C 180,E1 -6217.339,E2 -6217.339} C_VEL
LIN {X 0,Y 495.287,Z 538.301,A -85,B 0,C 180,E1 -6218.98,E2 -6218.98} C_VEL
LIN {X 0,Y 495.595,Z 530.463,A -85,B 0,C 180,E1 -6220.623,E2 -6220.623} C_VEL
LIN {X 0,Y 495.824,Z 522.351,A -85,B 0,C 180,E1 -6222.032,E2 -6222.032} C_VEL
LIN {X 0,Y 496.386,Z 512.087,A -85,B 0,C 180,E1 -6223.51,E2 -6223.51} C_VEL
LIN {X 0,Y 496.875,Z 501.818,A -85,B 0,C 180,E1 -6224.749,E2 -6224.749} C_VEL
LIN {X 0,Y 497.557,Z 489.185,A -85,B 0,C 180,E1 -6226.026,E2 -6226.026} C_VEL
LIN {X 0,Y 498.243,Z 475.983,A -85,B 0,C 180,E1 -6227.124,E2 -6227.124} C_VEL
LIN {X 0,Y 498.956,Z 462.344,A -85,B 0,C 180,E1 -6228.052,E2 -6228.052} C_VEL
LIN {X 0,Y 499.547,Z 448.22,A -85,B 0,C 180,E1 -6228.826,E2 -6228.826} C_VEL
LIN {X 0,Y 500.145,Z 432.917,A -85,B 0,C 180,E1 -6229.47,E2 -6229.47} C_VEL
LIN {X 0,Y 500.609,Z 417.813,A -85,B 0,C 180,E1 -6229.93,E2 -6229.93} C_VEL
LIN {X 0,Y 500.879,Z 401.928,A -85,B 0,C 180,E1 -6230.24,E2 -6230.24} C_VEL
LIN {X 0,Y 502.052,Z 262.884,A -85,B 0,C 180,E1 -6232.279,E2 -6232.279} C_VEL
LIN {X 0,Y 498.342,Z 244.001,A -85,B 0,C 180,E1 -6232.744,E2 -6232.744} C_VEL
LIN {X 0,Y 499.355,Z 221.505,A -85,B 0,C 180,E1 -6235.867,E2 -6235.867} C_VEL
LIN {X 0,Y 499.506,Z 216.781,A -85,B 0,C 180,E1 -6236.533,E2 -6236.533} C_VEL
LIN {X 0,Y 496.827,Z 204.518,A -85,B 0,C 180,E1 -6238.454,E2 -6238.454} C_VEL
LIN {X 0,Y 495.796,Z 200.351,A -85,B 0,C 180,E1 -6239.161,E2 -6239.161} C_VEL
LIN {X 0,Y 495.765,Z 200.349,A -85,B 0,C 180,E1 -6242.594,E2 -6242.594} C_VEL
LIN {X 0,Y 495.752,Z 200.353,A -85,B 0,C 180,E1 -6245.536,E2 -6245.536} C_VEL
LIN {X 0,Y 495.765,Z 200.353,A -85,B 0,C 180,E1 -6248.768,E2 -6248.768} C_VEL
LIN {X 0,Y 495.756,Z 200.357,A -85,B 0,C 180,E1 -6251.78,E2 -6251.78} C_VEL
LIN {X 0,Y 495.744,Z 200.353,A -85,B 0,C 180,E1 -6255.139,E2 -6255.139} C_VEL
LIN {X 0,Y 495.755,Z 200.356,A -85,B 0,C 180,E1 -6258.219,E2 -6258.219} C_VEL
LIN {X 0,Y 495.762,Z 200.351,A -85,B 0,C 180,E1 -6261.23,E2 -6261.23} C_VEL
LIN {X 0,Y 495.751,Z 200.351,A -85,B 0,C 180,E1 -6264.463,E2 -6264.463} C_VEL
LIN {X 0,Y 495.762,Z 200.352,A -85,B 0,C 180,E1 -6267.405,E2 -6267.405} C_VEL
LIN {X 0,Y 495.774,Z 200.351,A -85,B 0,C 180,E1 -6270.254,E2 -6270.254} C_VEL
LIN {X 0,Y 495.815,Z 200.346,A -85,B 0,C 180,E1 -6273.25,E2 -6273.25} C_VEL
LIN {X 0,Y 495.744,Z 200.359,A -85,B 0,C 180,E1 -6275.725,E2 -6275.725} C_VEL
LIN {X 0,Y 495.738,Z 200.346,A -85,B 0,C 180,E1 -6278.371,E2 -6278.371} C_VEL
LIN {X 0,Y 495.776,Z 200.35,A -85,B 0,C 180,E1 -6280.971,E2 -6280.971} C_VEL
LIN {X 0,Y 495.772,Z 200.355,A -85,B 0,C 180,E1 -6283.53,E2 -6283.53} C_VEL
LIN {X 0,Y 495.785,Z 200.35,A -85,B 0,C 180,E1 -6286.055,E2 -6286.055} C_VEL
LIN {X 0,Y 495.845,Z 200.34,A -85,B 0,C 180,E1 -6288.555,E2 -6288.555} C_VEL
LIN {X 0,Y 495.864,Z 200.341,A -85,B 0,C 180,E1 -6291.852,E2 -6291.852} C_VEL
LIN {X 0,Y 495.888,Z 200.336,A -85,B 0,C 180,E1 -6294.307,E2 -6294.307} C_VEL
LIN {X 0,Y 495.984,Z 200.33,A -85,B 0,C 180,E1 -6297.564,E2 -6297.564} C_VEL
LIN {X 0,Y 495.987,Z 200.322,A -85,B 0,C 180,E1 -6300,E2 -6300} C_VEL
LIN {X 0,Y 495.984,Z 200.324,A -85,B 0,C 180,E1 -6302.436,E2 -6302.436} C_VEL
LIN {X 0,Y 495.895,Z 200.338,A -85,B 0,C 180,E1 -6305.694,E2 -6305.694} C_VEL
LIN {X 0,Y 495.865,Z 200.336,A -85,B 0,C 180,E1 -6308.148,E2 -6308.148} C_VEL
LIN {X 0,Y 495.846,Z 200.345,A -85,B 0,C 180,E1 -6311.445,E2 -6311.445} C_VEL
LIN {X 0,Y 495.781,Z 200.352,A -85,B 0,C 180,E1 -6314.783,E2 -6314.783} C_VEL
LIN {X 0,Y 495.78,Z 200.355,A -85,B 0,C 180,E1 -6317.319,E2 -6317.319} C_VEL
LIN {X 0,Y 495.763,Z 200.35,A -85,B 0,C 180,E1 -6319.891,E2 -6319.891} C_VEL
LIN {X 0,Y 495.753,Z 200.358,A -85,B 0,C 180,E1 -6322.862,E2 -6322.862} C_VEL
LIN {X 0,Y 495.783,Z 200.337,A -85,B 0,C 180,E1 -6326.068,E2 -6326.068} C_VEL
LIN {X 0,Y 495.773,Z 200.354,A -85,B 0,C 180,E1 -6328.815,E2 -6328.815} C_VEL
LIN {X 0,Y 495.752,Z 200.353,A -85,B 0,C 180,E1 -6331.727,E2 -6331.727} C_VEL
LIN {X 0,Y 495.77,Z 200.354,A -85,B 0,C 180,E1 -6334.696,E2 -6334.696} C_VEL
LIN {X 0,Y 495.726,Z 200.356,A -85,B 0,C 180,E1 -6337.562,E2 -6337.562} C_VEL
LIN {X 0,Y 495.762,Z 200.356,A -85,B 0,C 180,E1 -6340.701,E2 -6340.701} C_VEL
LIN {X 0,Y 495.732,Z 200.355,A -85,B 0,C 180,E1 -6344.001,E2 -6344.001} C_VEL
LIN {X 0,Y 495.73,Z 200.36,A -85,B 0,C 180,E1 -6347.119,E2 -6347.119} C_VEL
LIN {X 0,Y 495.755,Z 200.354,A -85,B 0,C 180,E1 -6349.954,E2 -6349.954} C_VEL
LIN {X 0,Y 495.725,Z 200.363,A -85,B 0,C 180,E1 -6352.554,E2 -6352.554} C_VEL
LIN {X 0,Y 495.775,Z 200.352,A -85,B 0,C 180,E1 -6355.457,E2 -6355.457} C_VEL
LIN {X 0,Y 495.755,Z 200.359,A -85,B 0,C 180,E1 -6358.365,E2 -6358.365} C_VEL
LIN {X 0,Y 495.752,Z 200.357,A -85,B 0,C 180,E1 -6360.768,E2 -6360.768} C_VEL
LIN {X 0,Y 495.097,Z 200.44,A -85,B 0,C 180,E1 -6361.221,E2 -6361.221} C_VEL
LIN {X 0,Y 492.308,Z 200.789,A -85,B 0,C 180,E1 -6361.93,E2 -6361.93} C_VEL
LIN {X 0,Y 489.481,Z 201.142,A -85,B 0,C 180,E1 -6362.647,E2 -6362.647} C_VEL
LIN {X 0,Y 488.787,Z 201.227,A -85,B 0,C 180,E1 -6363.108,E2 -6363.108} C_VEL
LIN {X 0,Y 488.793,Z 201.398,A -85,B 0,C 180,E1 -6363.875,E2 -6363.875} C_VEL
LIN {X 0,Y 491.594,Z 214.228,A -85,B 0,C 180,E1 -6366.201,E2 -6366.201} C_VEL
LIN {X 0,Y 491.69,Z 218.973,A -85,B 0,C 180,E1 -6366.986,E2 -6366.986} C_VEL
LIN {X 0,Y 495.649,Z 236.62,A -85,B 0,C 180,E1 -6367.461,E2 -6367.461} C_VEL
LIN {X 0,Y 494.603,Z 351.118,A -85,B 0,C 180,E1 -6369.165,E2 -6369.165} C_VEL
LIN {X 0,Y 494.197,Z 385.376,A -85,B 0,C 180,E1 -6369.702,E2 -6369.702} C_VEL
LIN {X 0,Y 493.892,Z 400.333,A -85,B 0,C 180,E1 -6370.101,E2 -6370.101} C_VEL
LIN {X 0,Y 493.364,Z 415.222,A -85,B 0,C 180,E1 -6370.665,E2 -6370.665} C_VEL
LIN {X 0,Y 492.776,Z 429.677,A -85,B 0,C 180,E1 -6371.391,E2 -6371.391} C_VEL
LIN {X 0,Y 492.096,Z 442.939,A -85,B 0,C 180,E1 -6372.226,E2 -6372.226} C_VEL
LIN {X 0,Y 491.34,Z 456.415,A -85,B 0,C 180,E1 -6373.27,E2 -6373.27} C_VEL
LIN {X 0,Y 490.637,Z 468.632,A -85,B 0,C 180,E1 -6374.421,E2 -6374.421} C_VEL
LIN {X 0,Y 489.988,Z 479.757,A -85,B 0,C 180,E1 -6375.675,E2 -6375.675} C_VEL
LIN {X 0,Y 489.36,Z 490.563,A -85,B 0,C 180,E1 -6377.138,E2 -6377.138} C_VEL
LIN {X 0,Y 488.933,Z 499.525,A -85,B 0,C 180,E1 -6378.601,E2 -6378.601} C_VEL
LIN {X 0,Y 488.542,Z 506.954,A -85,B 0,C 180,E1 -6380.06,E2 -6380.06} C_VEL
LIN {X 0,Y 488.293,Z 513.897,A -85,B 0,C 180,E1 -6381.725,E2 -6381.725} C_VEL
LIN {X 0,Y 488.089,Z 519.636,A -85,B 0,C 180,E1 -6383.48,E2 -6383.48} C_VEL
LIN {X 0,Y 487.949,Z 523.479,A -85,B 0,C 180,E1 -6385.042,E2 -6385.042} C_VEL
LIN {X 0,Y 487.96,Z 526.375,A -85,B 0,C 180,E1 -6386.697,E2 -6386.697} C_VEL
LIN {X 0,Y 487.89,Z 528.123,A -85,B 0,C 180,E1 -6388.349,E2 -6388.349} C_VEL
LIN {X 0,Y 487.817,Z 528.737,A -85,B 0,C 180,E1 -6390,E2 -6390} C_VEL
LIN {X 0,Y 487.891,Z 528.177,A -85,B 0,C 180,E1 -6391.651,E2 -6391.651} C_VEL
LIN {X 0,Y 487.96,Z 526.502,A -85,B 0,C 180,E1 -6393.303,E2 -6393.303} C_VEL
LIN {X 0,Y 487.946,Z 523.674,A -85,B 0,C 180,E1 -6394.958,E2 -6394.958} C_VEL
LIN {X 0,Y 488.097,Z 519.619,A -85,B 0,C 180,E1 -6396.614,E2 -6396.614} C_VEL
LIN {X 0,Y 488.292,Z 514.242,A -85,B 0,C 180,E1 -6398.275,E2 -6398.275} C_VEL
LIN {X 0,Y 488.511,Z 507.391,A -85,B 0,C 180,E1 -6399.941,E2 -6399.941} C_VEL
LIN {X 0,Y 488.91,Z 500.017,A -85,B 0,C 180,E1 -6401.4,E2 -6401.4} C_VEL
LIN {X 0,Y 489.335,Z 491.138,A -85,B 0,C 180,E1 -6402.862,E2 -6402.862} C_VEL
LIN {X 0,Y 489.853,Z 482.082,A -85,B 0,C 180,E1 -6404.117,E2 -6404.117} C_VEL
LIN {X 0,Y 490.46,Z 471.397,A -85,B 0,C 180,E1 -6405.372,E2 -6405.372} C_VEL
LIN {X 0,Y 491.121,Z 459.897,A -85,B 0,C 180,E1 -6406.508,E2 -6406.508} C_VEL
LIN {X 0,Y 491.85,Z 446.989,A -85,B 0,C 180,E1 -6407.569,E2 -6407.569} C_VEL
LIN {X 0,Y 492.601,Z 432.925,A -85,B 0,C 180,E1 -6408.508,E2 -6408.508} C_VEL
LIN {X 0,Y 493.201,Z 419.434,A -85,B 0,C 180,E1 -6409.23,E2 -6409.23} C_VEL
LIN {X 0,Y 493.756,Z 404.364,A -85,B 0,C 180,E1 -6409.851,E2 -6409.851} C_VEL
LIN {X 0,Y 494.116,Z 389.874,A -85,B 0,C 180,E1 -6410.284,E2 -6410.284} C_VEL
LIN {X 0,Y 494.376,Z 374.969,A -85,B 0,C 180,E1 -6410.572,E2 -6410.572} C_VEL
LIN {X 0,Y 495.712,Z 237.618,A -85,B 0,C 180,E1 -6412.612,E2 -6412.612} C_VEL
LIN {X 0,Y 493.016,Z 224.776,A -85,B 0,C 180,E1 -6412.943,E2 -6412.943} C_VEL
LIN {X 0,Y 491.681,Z 218.954,A -85,B 0,C 180,E1 -6413.108,E2 -6413.108} C_VEL
LIN {X 0,Y 491.699,Z 214.583,A -85,B 0,C 180,E1 -6413.827,E2 -6413.827} C_VEL
LIN {X 0,Y 488.773,Z 201.229,A -85,B 0,C 180,E1 -6416.269,E2 -6416.269} C_VEL
LIN {X 0,Y 488.722,Z 201.235,A -85,B 0,C 180,E1 -6419.27,E2 -6419.27} C_VEL
LIN {X 0,Y 488.702,Z 201.235,A -85,B 0,C 180,E1 -6422.146,E2 -6422.146} C_VEL
LIN {X 0,Y 488.719,Z 201.235,A -85,B 0,C 180,E1 -6425.114,E2 -6425.114} C_VEL
LIN {X 0,Y 488.678,Z 201.238,A -85,B 0,C 180,E1 -6428.199,E2 -6428.199} C_VEL
LIN {X 0,Y 488.716,Z 201.238,A -85,B 0,C 180,E1 -6431.414,E2 -6431.414} C_VEL
LIN {X 0,Y 488.698,Z 201.232,A -85,B 0,C 180,E1 -6434.023,E2 -6434.023} C_VEL
LIN {X 0,Y 488.705,Z 201.232,A -85,B 0,C 180,E1 -6437.173,E2 -6437.173} C_VEL
LIN {X 0,Y 488.727,Z 201.231,A -85,B 0,C 180,E1 -6439.676,E2 -6439.676} C_VEL
LIN {X 0,Y 488.673,Z 201.228,A -85,B 0,C 180,E1 -6442.277,E2 -6442.277} C_VEL
LIN {X 0,Y 488.722,Z 201.234,A -85,B 0,C 180,E1 -6445.051,E2 -6445.051} C_VEL
LIN {X 0,Y 488.699,Z 201.223,A -85,B 0,C 180,E1 -6448.045,E2 -6448.045} C_VEL
LIN {X 0,Y 488.727,Z 201.228,A -85,B 0,C 180,E1 -6450.73,E2 -6450.73} C_VEL
LIN {X 0,Y 488.749,Z 201.225,A -85,B 0,C 180,E1 -6453.527,E2 -6453.527} C_VEL
LIN {X 0,Y 488.684,Z 201.234,A -85,B 0,C 180,E1 -6456.254,E2 -6456.254} C_VEL
LIN {X 0,Y 488.737,Z 201.232,A -85,B 0,C 180,E1 -6459.175,E2 -6459.175} C_VEL
LIN {X 0,Y 488.75,Z 201.223,A -85,B 0,C 180,E1 -6461.627,E2 -6461.627} C_VEL
LIN {X 0,Y 488.753,Z 201.227,A -85,B 0,C 180,E1 -6464.999,E2 -6464.999} C_VEL
LIN {X 0,Y 488.799,Z 201.222,A -85,B 0,C 180,E1 -6468.387,E2 -6468.387} C_VEL
LIN {X 0,Y 488.808,Z 201.217,A -85,B 0,C 180,E1 -6471.733,E2 -6471.733} C_VEL
LIN {X 0,Y 488.847,Z 201.214,A -85,B 0,C 180,E1 -6474.224,E2 -6474.224} C_VEL
LIN {X 0,Y 488.952,Z 201.2,A -85,B 0,C 180,E1 -6477.529,E2 -6477.529} C_VEL
LIN {X 0,Y 488.958,Z 201.196,A -85,B 0,C 180,E1 -6480,E2 -6480} C_VEL
LIN {X 0,Y 488.952,Z 201.206,A -85,B 0,C 180,E1 -6482.471,E2 -6482.471} C_VEL
LIN {X 0,Y 488.847,Z 201.213,A -85,B 0,C 180,E1 -6485.776,E2 -6485.776} C_VEL
LIN {X 0,Y 488.809,Z 201.221,A -85,B 0,C 180,E1 -6488.266,E2 -6488.266} C_VEL
LIN {X 0,Y 488.798,Z 201.22,A -85,B 0,C 180,E1 -6491.613,E2 -6491.613} C_VEL
LIN {X 0,Y 488.755,Z 201.227,A -85,B 0,C 180,E1 -6495,E2 -6495} C_VEL
LIN {X 0,Y 488.746,Z 201.232,A -85,B 0,C 180,E1 -6498.442,E2 -6498.442} C_VEL
LIN {X 0,Y 488.699,Z 201.23,A -85,B 0,C 180,E1 -6501.071,E2 -6501.071} C_VEL
LIN {X 0,Y 488.685,Z 201.236,A -85,B 0,C 180,E1 -6503.746,E2 -6503.746} C_VEL
LIN {X 0,Y 488.784,Z 201.223,A -85,B 0,C 180,E1 -6506.944,E2 -6506.944} C_VEL
LIN {X 0,Y 488.726,Z 201.235,A -85,B 0,C 180,E1 -6510.219,E2 -6510.219} C_VEL
LIN {X 0,Y 488.728,Z 201.226,A -85,B 0,C 180,E1 -6513.485,E2 -6513.485} C_VEL
LIN {X 0,Y 488.682,Z 201.238,A -85,B 0,C 180,E1 -6516.356,E2 -6516.356} C_VEL
LIN {X 0,Y 488.694,Z 201.23,A -85,B 0,C 180,E1 -6519.255,E2 -6519.255} C_VEL
LIN {X 0,Y 488.702,Z 201.227,A -85,B 0,C 180,E1 -6521.601,E2 -6521.601} C_VEL
LIN {X 0,Y 488.706,Z 201.232,A -85,B 0,C 180,E1 -6524.802,E2 -6524.802} C_VEL
LIN {X 0,Y 488.686,Z 201.236,A -85,B 0,C 180,E1 -6527.475,E2 -6527.475} C_VEL
LIN {X 0,Y 488.729,Z 201.233,A -85,B 0,C 180,E1 -6529.677,E2 -6529.677} C_VEL
LIN {X 0,Y 488.676,Z 201.234,A -85,B 0,C 180,E1 -6532.278,E2 -6532.278} C_VEL
LIN {X 0,Y 488.724,Z 201.231,A -85,B 0,C 180,E1 -6535.052,E2 -6535.052} C_VEL
LIN {X 0,Y 488.701,Z 201.238,A -85,B 0,C 180,E1 -6538.046,E2 -6538.046} C_VEL
LIN {X 0,Y 488.767,Z 201.33,A -85,B 0,C 180,E1 -6540.586,E2 -6540.586} C_VEL
LIN {X 0,Y 492.38,Z 216.593,A -85,B 0,C 180,E1 -6543.053,E2 -6543.053} C_VEL
LIN {X 0,Y 492.664,Z 219.75,A -85,B 0,C 180,E1 -6543.527,E2 -6543.527} C_VEL
LIN {X 0,Y 491.638,Z 241.718,A -85,B 0,C 180,E1 -6546.629,E2 -6546.629} C_VEL
LIN {X 0,Y 491.532,Z 243.795,A -85,B 0,C 180,E1 -6546.921,E2 -6546.921} C_VEL
LIN {X 0,Y 495.47,Z 263.791,A -85,B 0,C 180,E1 -6547.426,E2 -6547.426} C_VEL
LIN {X 0,Y 494.263,Z 396.401,A -85,B 0,C 180,E1 -6549.396,E2 -6549.396} C_VEL
LIN {X 0,Y 494.016,Z 414.207,A -85,B 0,C 180,E1 -6549.711,E2 -6549.711} C_VEL
LIN {X 0,Y 493.56,Z 429.055,A -85,B 0,C 180,E1 -6550.13,E2 -6550.13} C_VEL
LIN {X 0,Y 493.046,Z 443.117,A -85,B 0,C 180,E1 -6550.682,E2 -6550.682} C_VEL
LIN {X 0,Y 492.362,Z 456.84,A -85,B 0,C 180,E1 -6551.375,E2 -6551.375} C_VEL
LIN {X 0,Y 491.77,Z 470.059,A -85,B 0,C 180,E1 -6552.214,E2 -6552.214} C_VEL
LIN {X 0,Y 490.985,Z 483.516,A -85,B 0,C 180,E1 -6553.258,E2 -6553.258} C_VEL
LIN {X 0,Y 490.308,Z 495.776,A -85,B 0,C 180,E1 -6554.41,E2 -6554.41} C_VEL
LIN {X 0,Y 489.665,Z 506.971,A -85,B 0,C 180,E1 -6555.666,E2 -6555.666} C_VEL
LIN {X 0,Y 489.046,Z 517.836,A -85,B 0,C 180,E1 -6557.13,E2 -6557.13} C_VEL
LIN {X 0,Y 488.65,Z 526.889,A -85,B 0,C 180,E1 -6558.594,E2 -6558.594} C_VEL
LIN {X 0,Y 488.315,Z 534.397,A -85,B 0,C 180,E1 -6560.055,E2 -6560.055} C_VEL
LIN {X 0,Y 488.12,Z 541.406,A -85,B 0,C 180,E1 -6561.722,E2 -6561.722} C_VEL
LIN {X 0,Y 487.998,Z 547.484,A -85,B 0,C 180,E1 -6563.573,E2 -6563.573} C_VEL
LIN {X 0,Y 487.926,Z 551.083,A -85,B 0,C 180,E1 -6565.042,E2 -6565.042} C_VEL
LIN {X 0,Y 487.942,Z 554.005,A -85,B 0,C 180,E1 -6566.697,E2 -6566.697} C_VEL
LIN {X 0,Y 487.888,Z 555.747,A -85,B 0,C 180,E1 -6568.349,E2 -6568.349} C_VEL
LIN {X 0,Y 487.816,Z 556.342,A -85,B 0,C 180,E1 -6570,E2 -6570} C_VEL
LIN {X 0,Y 487.888,Z 555.744,A -85,B 0,C 180,E1 -6571.651,E2 -6571.651} C_VEL
LIN {X 0,Y 487.942,Z 554,A -85,B 0,C 180,E1 -6573.303,E2 -6573.303} C_VEL
LIN {X 0,Y 487.927,Z 551.081,A -85,B 0,C 180,E1 -6574.958,E2 -6574.958} C_VEL
LIN {X 0,Y 488.069,Z 546.923,A -85,B 0,C 180,E1 -6576.615,E2 -6576.615} C_VEL
LIN {X 0,Y 488.12,Z 541.407,A -85,B 0,C 180,E1 -6578.278,E2 -6578.278} C_VEL
LIN {X 0,Y 488.315,Z 534.391,A -85,B 0,C 180,E1 -6579.945,E2 -6579.945} C_VEL
LIN {X 0,Y 488.655,Z 526.885,A -85,B 0,C 180,E1 -6581.406,E2 -6581.406} C_VEL
LIN {X 0,Y 489.046,Z 517.837,A -85,B 0,C 180,E1 -6582.87,E2 -6582.87} C_VEL
LIN {X 0,Y 489.672,Z 506.97,A -85,B 0,C 180,E1 -6584.334,E2 -6584.334} C_VEL
LIN {X 0,Y 490.37,Z 494.757,A -85,B 0,C 180,E1 -6585.695,E2 -6585.695} C_VEL
LIN {X 0,Y 491.053,Z 482.304,A -85,B 0,C 180,E1 -6586.847,E2 -6586.847} C_VEL
LIN {X 0,Y 491.748,Z 470.052,A -85,B 0,C 180,E1 -6587.787,E2 -6587.787} C_VEL
LIN {X 0,Y 492.367,Z 456.825,A -85,B 0,C 180,E1 -6588.625,E2 -6588.625} C_VEL
LIN {X 0,Y 493.09,Z 443.039,A -85,B 0,C 180,E1 -6589.32,E2 -6589.32} C_VEL
LIN {X 0,Y 493.599,Z 428.247,A -85,B 0,C 180,E1 -6589.898,E2 -6589.898} C_VEL
LIN {X 0,Y 494.019,Z 413.387,A -85,B 0,C 180,E1 -6590.308,E2 -6590.308} C_VEL
LIN {X 0,Y 494.275,Z 392.771,A -85,B 0,C 180,E1 -6590.658,E2 -6590.658} C_VEL
LIN {X 0,Y 495.514,Z 264.186,A -85,B 0,C 180,E1 -6592.565,E2 -6592.565} C_VEL
LIN {X 0,Y 491.537,Z 243.788,A -85,B 0,C 180,E1 -6593.078,E2 -6593.078} C_VEL
LIN {X 0,Y 492.587,Z 221.311,A -85,B 0,C 180,E1 -6596.25,E2 -6596.25} C_VEL
LIN {X 0,Y 492.637,Z 218.162,A -85,B 0,C 180,E1 -6596.703,E2 -6596.703} C_VEL
LIN {X 0,Y 489.87,Z 205.796,A -85,B 0,C 180,E1 -6598.677,E2 -6598.677} C_VEL
LIN {X 0,Y 488.727,Z 201.232,A -85,B 0,C 180,E1 -6599.447,E2 -6599.447} C_VEL
LIN {X 0,Y 488.701,Z 201.234,A -85,B 0,C 180,E1 -6602.146,E2 -6602.146} C_VEL
LIN {X 0,Y 488.718,Z 201.227,A -85,B 0,C 180,E1 -6605.114,E2 -6605.114} C_VEL
LIN {X 0,Y 488.679,Z 201.241,A -85,B 0,C 180,E1 -6608.199,E2 -6608.199} C_VEL
LIN {X 0,Y 488.745,Z 201.231,A -85,B 0,C 180,E1 -6610.348,E2 -6610.348} C_VEL
LIN {X 0,Y 488.682,Z 201.237,A -85,B 0,C 180,E1 -6613.654,E2 -6613.654} C_VEL
LIN {X 0,Y 488.681,Z 201.236,A -85,B 0,C 180,E1 -6616.345,E2 -6616.345} C_VEL
LIN {X 0,Y 488.727,Z 201.231,A -85,B 0,C 180,E1 -6619.676,E2 -6619.676} C_VEL
LIN {X 0,Y 488.674,Z 201.236,A -85,B 0,C 180,E1 -6622.277,E2 -6622.277} C_VEL
LIN {X 0,Y 488.721,Z 201.226,A -85,B 0,C 180,E1 -6625.051,E2 -6625.051} C_VEL
LIN {X 0,Y 488.699,Z 201.235,A -85,B 0,C 180,E1 -6628.045,E2 -6628.045} C_VEL
LIN {X 0,Y 488.726,Z 201.226,A -85,B 0,C 180,E1 -6630.73,E2 -6630.73} C_VEL
LIN {X 0,Y 488.749,Z 201.229,A -85,B 0,C 180,E1 -6633.528,E2 -6633.528} C_VEL
LIN {X 0,Y 488.685,Z 201.232,A -85,B 0,C 180,E1 -6636.254,E2 -6636.254} C_VEL
LIN {X 0,Y 488.737,Z 201.219,A -85,B 0,C 180,E1 -6639.175,E2 -6639.175} C_VEL
LIN {X 0,Y 488.75,Z 201.233,A -85,B 0,C 180,E1 -6641.627,E2 -6641.627} C_VEL
LIN {X 0,Y 488.753,Z 201.225,A -85,B 0,C 180,E1 -6644.999,E2 -6644.999} C_VEL
LIN {X 0,Y 488.799,Z 201.218,A -85,B 0,C 180,E1 -6648.387,E2 -6648.387} C_VEL
LIN {X 0,Y 488.809,Z 201.222,A -85,B 0,C 180,E1 -6651.734,E2 -6651.734} C_VEL
LIN {X 0,Y 488.847,Z 201.213,A -85,B 0,C 180,E1 -6654.224,E2 -6654.224} C_VEL
LIN {X 0,Y 488.952,Z 201.207,A -85,B 0,C 180,E1 -6657.529,E2 -6657.529} C_VEL
LIN {X 0,Y 488.959,Z 201.197,A -85,B 0,C 180,E1 -6660,E2 -6660} C_VEL
LIN {X 0,Y 488.952,Z 201.2,A -85,B 0,C 180,E1 -6662.471,E2 -6662.471} C_VEL
LIN {X 0,Y 488.853,Z 201.215,A -85,B 0,C 180,E1 -6665.776,E2 -6665.776} C_VEL
LIN {X 0,Y 488.809,Z 201.215,A -85,B 0,C 180,E1 -6668.267,E2 -6668.267} C_VEL
LIN {X 0,Y 488.799,Z 201.22,A -85,B 0,C 180,E1 -6671.613,E2 -6671.613} C_VEL
LIN {X 0,Y 488.753,Z 201.23,A -85,B 0,C 180,E1 -6675.001,E2 -6675.001} C_VEL
LIN {X 0,Y 488.746,Z 201.226,A -85,B 0,C 180,E1 -6678.443,E2 -6678.443} C_VEL
LIN {X 0,Y 488.698,Z 201.236,A -85,B 0,C 180,E1 -6681.071,E2 -6681.071} C_VEL
LIN {X 0,Y 488.684,Z 201.232,A -85,B 0,C 180,E1 -6683.746,E2 -6683.746} C_VEL
LIN {X 0,Y 488.784,Z 201.216,A -85,B 0,C 180,E1 -6686.944,E2 -6686.944} C_VEL
LIN {X 0,Y 488.727,Z 201.228,A -85,B 0,C 180,E1 -6690.219,E2 -6690.219} C_VEL
LIN {X 0,Y 488.729,Z 201.227,A -85,B 0,C 180,E1 -6693.485,E2 -6693.485} C_VEL
LIN {X 0,Y 488.683,Z 201.235,A -85,B 0,C 180,E1 -6696.356,E2 -6696.356} C_VEL
LIN {X 0,Y 488.696,Z 201.233,A -85,B 0,C 180,E1 -6699.255,E2 -6699.255} C_VEL
LIN {X 0,Y 488.703,Z 201.229,A -85,B 0,C 180,E1 -6701.601,E2 -6701.601} C_VEL
LIN {X 0,Y 488.697,Z 201.231,A -85,B 0,C 180,E1 -6704.025,E2 -6704.025} C_VEL
LIN {X 0,Y 488.712,Z 201.234,A -85,B 0,C 180,E1 -6707.173,E2 -6707.173} C_VEL
LIN {X 0,Y 488.729,Z 201.229,A -85,B 0,C 180,E1 -6709.677,E2 -6709.677} C_VEL
LIN {X 0,Y 488.676,Z 201.241,A -85,B 0,C 180,E1 -6712.842,E2 -6712.842} C_VEL
LIN {X 0,Y 488.728,Z 201.23,A -85,B 0,C 180,E1 -6715.888,E2 -6715.888} C_VEL
LIN {X 0,Y 488.691,Z 201.237,A -85,B 0,C 180,E1 -6718.821,E2 -6718.821} C_VEL
LIN {X 0,Y 488.744,Z 201.231,A -85,B 0,C 180,E1 -6721.672,E2 -6721.672} C_VEL
LIN {X 0,Y 488.787,Z 201.227,A -85,B 0,C 180,E1 -6723.108,E2 -6723.108} C_VEL
LIN {X 0,Y 488.562,Z 201.788,A -85,B 0,C 180,E1 -6723.561,E2 -6723.561} C_VEL
LIN {X 0,Y 488.067,Z 203.199,A -85,B 0,C 180,E1 -6723.989,E2 -6723.989} C_VEL
LIN {X 0,Y 486.675,Z 207.441,A -85,B 0,C 180,E1 -6724.776,E2 -6724.776} C_VEL
LIN {X 0,Y 484.937,Z 214.724,A -85,B 0,C 180,E1 -6725.903,E2 -6725.903} C_VEL
LIN {X 0,Y 484.857,Z 217.051,A -85,B 0,C 180,E1 -6726.289,E2 -6726.289} C_VEL
LIN {X 0,Y 484.928,Z 219.5,A -85,B 0,C 180,E1 -6726.657,E2 -6726.657} C_VEL
LIN {X 0,Y 489.096,Z 237.386,A -85,B 0,C 180,E1 -6727.15,E2 -6727.15} C_VEL
LIN {X 0,Y 487.995,Z 351.349,A -85,B 0,C 180,E1 -6728.87,E2 -6728.87} C_VEL
LIN {X 0,Y 487.567,Z 385.596,A -85,B 0,C 180,E1 -6729.414,E2 -6729.414} C_VEL
LIN {X 0,Y 487.221,Z 400.851,A -85,B 0,C 180,E1 -6729.828,E2 -6729.828} C_VEL
LIN {X 0,Y 486.67,Z 415.574,A -85,B 0,C 180,E1 -6730.395,E2 -6730.395} C_VEL
LIN {X 0,Y 486.05,Z 429.886,A -85,B 0,C 180,E1 -6731.124,E2 -6731.124} C_VEL
LIN {X 0,Y 485.335,Z 443.147,A -85,B 0,C 180,E1 -6731.97,E2 -6731.97} C_VEL
LIN {X 0,Y 484.521,Z 456.622,A -85,B 0,C 180,E1 -6733.028,E2 -6733.028} C_VEL
LIN {X 0,Y 483.76,Z 468.839,A -85,B 0,C 180,E1 -6734.193,E2 -6734.193} C_VEL
LIN {X 0,Y 483.073,Z 479.963,A -85,B 0,C 180,E1 -6735.466,E2 -6735.466} C_VEL
LIN {X 0,Y 482.406,Z 490.769,A -85,B 0,C 180,E1 -6736.95,E2 -6736.95} C_VEL
LIN {X 0,Y 481.943,Z 499.73,A -85,B 0,C 180,E1 -6738.433,E2 -6738.433} C_VEL
LIN {X 0,Y 481.504,Z 507.159,A -85,B 0,C 180,E1 -6739.913,E2 -6739.913} C_VEL
LIN {X 0,Y 481.236,Z 514.101,A -85,B 0,C 180,E1 -6741.603,E2 -6741.603} C_VEL
LIN {X 0,Y 481.031,Z 520.074,A -85,B 0,C 180,E1 -6743.465,E2 -6743.465} C_VEL
LIN {X 0,Y 480.884,Z 523.681,A -85,B 0,C 180,E1 -6744.969,E2 -6744.969} C_VEL
LIN {X 0,Y 480.886,Z 526.577,A -85,B 0,C 180,E1 -6746.649,E2 -6746.649} C_VEL
LIN {X 0,Y 480.821,Z 528.324,A -85,B 0,C 180,E1 -6748.325,E2 -6748.325} C_VEL
LIN {X 0,Y 480.741,Z 528.937,A -85,B 0,C 180,E1 -6750,E2 -6750} C_VEL
LIN {X 0,Y 480.822,Z 528.377,A -85,B 0,C 180,E1 -6751.675,E2 -6751.675} C_VEL
LIN {X 0,Y 480.887,Z 526.701,A -85,B 0,C 180,E1 -6753.351,E2 -6753.351} C_VEL
LIN {X 0,Y 480.88,Z 523.873,A -85,B 0,C 180,E1 -6755.031,E2 -6755.031} C_VEL
LIN {X 0,Y 481.041,Z 519.818,A -85,B 0,C 180,E1 -6756.712,E2 -6756.712} C_VEL
LIN {X 0,Y 481.235,Z 514.441,A -85,B 0,C 180,E1 -6758.397,E2 -6758.397} C_VEL
LIN {X 0,Y 481.479,Z 507.591,A -85,B 0,C 180,E1 -6760.088,E2 -6760.088} C_VEL
LIN {X 0,Y 481.921,Z 500.216,A -85,B 0,C 180,E1 -6761.567,E2 -6761.567} C_VEL
LIN {X 0,Y 482.38,Z 491.337,A -85,B 0,C 180,E1 -6763.051,E2 -6763.051} C_VEL
LIN {X 0,Y 482.928,Z 482.28,A -85,B 0,C 180,E1 -6764.323,E2 -6764.323} C_VEL
LIN {X 0,Y 483.578,Z 471.595,A -85,B 0,C 180,E1 -6765.596,E2 -6765.596} C_VEL
LIN {X 0,Y 484.262,Z 460.669,A -85,B 0,C 180,E1 -6766.695,E2 -6766.695} C_VEL
LIN {X 0,Y 484.984,Z 448.603,A -85,B 0,C 180,E1 -6767.717,E2 -6767.717} C_VEL
LIN {X 0,Y 485.778,Z 434.878,A -85,B 0,C 180,E1 -6768.668,E2 -6768.668} C_VEL
LIN {X 0,Y 486.404,Z 421.677,A -85,B 0,C 180,E1 -6769.409,E2 -6769.409} C_VEL
LIN {X 0,Y 486.985,Z 406.405,A -85,B 0,C 180,E1 -6770.072,E2 -6770.072} C_VEL
LIN {X 0,Y 487.436,Z 391.796,A -85,B 0,C 180,E1 -6770.532,E2 -6770.532} C_VEL
LIN {X 0,Y 487.747,Z 375.748,A -85,B 0,C 180,E1 -6770.855,E2 -6770.855} C_VEL
LIN {X 0,Y 489.128,Z 237.648,A -85,B 0,C 180,E1 -6772.936,E2 -6772.936} C_VEL
LIN {X 0,Y 484.921,Z 219.168,A -85,B 0,C 180,E1 -6773.446,E2 -6773.446} C_VEL
LIN {X 0,Y 484.6,Z 214.994,A -85,B 0,C 180,E1 -6774.162,E2 -6774.162} C_VEL
LIN {X 0,Y 481.753,Z 202.104,A -85,B 0,C 180,E1 -6776.565,E2 -6776.565} C_VEL
LIN {X 0,Y 481.678,Z 202.113,A -85,B 0,C 180,E1 -6779.74,E2 -6779.74} C_VEL
LIN {X 0,Y 481.671,Z 202.11,A -85,B 0,C 180,E1 -6782.673,E2 -6782.673} C_VEL
LIN {X 0,Y 481.639,Z 202.117,A -85,B 0,C 180,E1 -6785.708,E2 -6785.708} C_VEL
LIN {X 0,Y 481.668,Z 202.113,A -85,B 0,C 180,E1 -6788.858,E2 -6788.858} C_VEL
LIN {X 0,Y 481.659,Z 202.111,A -85,B 0,C 180,E1 -6791.913,E2 -6791.913} C_VEL
LIN {X 0,Y 481.656,Z 202.109,A -85,B 0,C 180,E1 -6794.456,E2 -6794.456} C_VEL
LIN {X 0,Y 481.644,Z 202.108,A -85,B 0,C 180,E1 -6797.839,E2 -6797.839} C_VEL
LIN {X 0,Y 481.705,Z 202.105,A -85,B 0,C 180,E1 -6800.646,E2 -6800.646} C_VEL
LIN {X 0,Y 481.637,Z 202.11,A -85,B 0,C 180,E1 -6804.29,E2 -6804.29} C_VEL
LIN {X 0,Y 481.666,Z 202.104,A -85,B 0,C 180,E1 -6807.325,E2 -6807.325} C_VEL
LIN {X 0,Y 481.681,Z 202.102,A -85,B 0,C 180,E1 -6810.259,E2 -6810.259} C_VEL
LIN {X 0,Y 481.738,Z 202.102,A -85,B 0,C 180,E1 -6813.111,E2 -6813.111} C_VEL
LIN {X 0,Y 481.668,Z 202.107,A -85,B 0,C 180,E1 -6815.886,E2 -6815.886} C_VEL
LIN {X 0,Y 481.694,Z 202.112,A -85,B 0,C 180,E1 -6819.027,E2 -6819.027} C_VEL
LIN {X 0,Y 481.699,Z 202.101,A -85,B 0,C 180,E1 -6822.158,E2 -6822.158} C_VEL
LIN {X 0,Y 481.733,Z 202.105,A -85,B 0,C 180,E1 -6824.775,E2 -6824.775} C_VEL
LIN {X 0,Y 481.744,Z 202.099,A -85,B 0,C 180,E1 -6828.215,E2 -6828.215} C_VEL
LIN {X 0,Y 481.754,Z 202.096,A -85,B 0,C 180,E1 -6831.611,E2 -6831.611} C_VEL
LIN {X 0,Y 481.808,Z 202.09,A -85,B 0,C 180,E1 -6834.139,E2 -6834.139} C_VEL
LIN {X 0,Y 481.919,Z 202.076,A -85,B 0,C 180,E1 -6837.492,E2 -6837.492} C_VEL
LIN {X 0,Y 481.93,Z 202.072,A -85,B 0,C 180,E1 -6840,E2 -6840} C_VEL
LIN {X 0,Y 481.919,Z 202.083,A -85,B 0,C 180,E1 -6842.507,E2 -6842.507} C_VEL
LIN {X 0,Y 481.808,Z 202.09,A -85,B 0,C 180,E1 -6845.86,E2 -6845.86} C_VEL
LIN {X 0,Y 481.755,Z 202.1,A -85,B 0,C 180,E1 -6848.388,E2 -6848.388} C_VEL
LIN {X 0,Y 481.743,Z 202.099,A -85,B 0,C 180,E1 -6851.785,E2 -6851.785} C_VEL
LIN {X 0,Y 481.735,Z 202.101,A -85,B 0,C 180,E1 -6855.224,E2 -6855.224} C_VEL
LIN {X 0,Y 481.703,Z 202.108,A -85,B 0,C 180,E1 -6858.722,E2 -6858.722} C_VEL
LIN {X 0,Y 481.638,Z 202.109,A -85,B 0,C 180,E1 -6861.395,E2 -6861.395} C_VEL
LIN {X 0,Y 481.669,Z 202.114,A -85,B 0,C 180,E1 -6864.113,E2 -6864.113} C_VEL
LIN {X 0,Y 481.739,Z 202.1,A -85,B 0,C 180,E1 -6867.14,E2 -6867.14} C_VEL
LIN {X 0,Y 481.68,Z 202.109,A -85,B 0,C 180,E1 -6869.741,E2 -6869.741} C_VEL
LIN {X 0,Y 481.666,Z 202.108,A -85,B 0,C 180,E1 -6872.675,E2 -6872.675} C_VEL
LIN {X 0,Y 481.636,Z 202.114,A -85,B 0,C 180,E1 -6875.71,E2 -6875.71} C_VEL
LIN {X 0,Y 481.664,Z 202.106,A -85,B 0,C 180,E1 -6878.86,E2 -6878.86} C_VEL
LIN {X 0,Y 481.647,Z 202.109,A -85,B 0,C 180,E1 -6881.914,E2 -6881.914} C_VEL
LIN {X 0,Y 481.654,Z 202.113,A -85,B 0,C 180,E1 -6884.458,E2 -6884.458} C_VEL
LIN {X 0,Y 481.644,Z 202.117,A -85,B 0,C 180,E1 -6887.84,E2 -6887.84} C_VEL
LIN {X 0,Y 481.71,Z 202.104,A -85,B 0,C 180,E1 -6890.647,E2 -6890.647} C_VEL
LIN {X 0,Y 481.638,Z 202.116,A -85,B 0,C 180,E1 -6894.292,E2 -6894.292} C_VEL
LIN {X 0,Y 481.669,Z 202.112,A -85,B 0,C 180,E1 -6897.326,E2 -6897.326} C_VEL
LIN {X 0,Y 481.701,Z 202.124,A -85,B 0,C 180,E1 -6900.261,E2 -6900.261} C_VEL
LIN {X 0,Y 485.481,Z 217.975,A -85,B 0,C 180,E1 -6902.871,E2 -6902.871} C_VEL
LIN {X 0,Y 485.87,Z 221.134,A -85,B 0,C 180,E1 -6903.359,E2 -6903.359} C_VEL
LIN {X 0,Y 484.737,Z 243.571,A -85,B 0,C 180,E1 -6906.575,E2 -6906.575} C_VEL
LIN {X 0,Y 488.969,Z 265.839,A -85,B 0,C 180,E1 -6907.143,E2 -6907.143} C_VEL
LIN {X 0,Y 487.459,Z 409.244,A -85,B 0,C 180,E1 -6909.315,E2 -6909.315} C_VEL
LIN {X 0,Y 486.991,Z 424.822,A -85,B 0,C 180,E1 -6909.708,E2 -6909.708} C_VEL
LIN {X 0,Y 486.476,Z 439.363,A -85,B 0,C 180,E1 -6910.245,E2 -6910.245} C_VEL
LIN {X 0,Y 485.821,Z 452.835,A -85,B 0,C 180,E1 -6910.896,E2 -6910.896} C_VEL
LIN {X 0,Y 485.174,Z 465.165,A -85,B 0,C 180,E1 -6911.636,E2 -6911.636} C_VEL
LIN {X 0,Y 484.386,Z 478.207,A -85,B 0,C 180,E1 -6912.588,E2 -6912.588} C_VEL
LIN {X 0,Y 483.684,Z 490.52,A -85,B 0,C 180,E1 -6913.676,E2 -6913.676} C_VEL
LIN {X 0,Y 482.974,Z 501.411,A -85,B 0,C 180,E1 -6914.816,E2 -6914.816} C_VEL
LIN {X 0,Y 482.43,Z 511.681,A -85,B 0,C 180,E1 -6916.092,E2 -6916.092} C_VEL
LIN {X 0,Y 481.883,Z 521.72,A -85,B 0,C 180,E1 -6917.577,E2 -6917.577} C_VEL
LIN {X 0,Y 481.555,Z 530.065,A -85,B 0,C 180,E1 -6919.063,E2 -6919.063} C_VEL
LIN {X 0,Y 481.167,Z 537.899,A -85,B 0,C 180,E1 -6920.755,E2 -6920.755} C_VEL
LIN {X 0,Y 480.986,Z 544.136,A -85,B 0,C 180,E1 -6922.444,E2 -6922.444} C_VEL
LIN {X 0,Y 480.878,Z 548.959,A -85,B 0,C 180,E1 -6924.128,E2 -6924.128} C_VEL
LIN {X 0,Y 480.773,Z 552.492,A -85,B 0,C 180,E1 -6925.809,E2 -6925.809} C_VEL
LIN {X 0,Y 480.818,Z 554.819,A -85,B 0,C 180,E1 -6927.487,E2 -6927.487} C_VEL
LIN {X 0,Y 480.757,Z 555.988,A -85,B 0,C 180,E1 -6929.162,E2 -6929.162} C_VEL
LIN {X 0,Y 480.757,Z 555.987,A -85,B 0,C 180,E1 -6930.838,E2 -6930.838} C_VEL
LIN {X 0,Y 480.818,Z 554.815,A -85,B 0,C 180,E1 -6932.513,E2 -6932.513} C_VEL
LIN {X 0,Y 480.773,Z 552.488,A -85,B 0,C 180,E1 -6934.191,E2 -6934.191} C_VEL
LIN {X 0,Y 480.892,Z 548.961,A -85,B 0,C 180,E1 -6935.872,E2 -6935.872} C_VEL
LIN {X 0,Y 480.986,Z 544.14,A -85,B 0,C 180,E1 -6937.556,E2 -6937.556} C_VEL
LIN {X 0,Y 481.167,Z 537.896,A -85,B 0,C 180,E1 -6939.245,E2 -6939.245} C_VEL
LIN {X 0,Y 481.552,Z 530.058,A -85,B 0,C 180,E1 -6940.937,E2 -6940.937} C_VEL
LIN {X 0,Y 481.799,Z 522.275,A -85,B 0,C 180,E1 -6942.333,E2 -6942.333} C_VEL
LIN {X 0,Y 482.431,Z 511.679,A -85,B 0,C 180,E1 -6943.908,E2 -6943.908} C_VEL
LIN {X 0,Y 483.013,Z 501.411,A -85,B 0,C 180,E1 -6945.183,E2 -6945.183} C_VEL
LIN {X 0,Y 483.684,Z 490.299,A -85,B 0,C 180,E1 -6946.346,E2 -6946.346} C_VEL
LIN {X 0,Y 484.434,Z 478.208,A -85,B 0,C 180,E1 -6947.41,E2 -6947.41} C_VEL
LIN {X 0,Y 485.234,Z 465.15,A -85,B 0,C 180,E1 -6948.362,E2 -6948.362} C_VEL
LIN {X 0,Y 485.836,Z 452.814,A -85,B 0,C 180,E1 -6949.104,E2 -6949.104} C_VEL
LIN {X 0,Y 486.547,Z 438.151,A -85,B 0,C 180,E1 -6949.802,E2 -6949.802} C_VEL
LIN {X 0,Y 487.037,Z 423.336,A -85,B 0,C 180,E1 -6950.334,E2 -6950.334} C_VEL
LIN {X 0,Y 487.497,Z 407.706,A -85,B 0,C 180,E1 -6950.71,E2 -6950.71} C_VEL
LIN {X 0,Y 488.981,Z 266.033,A -85,B 0,C 180,E1 -6952.852,E2 -6952.852} C_VEL
LIN {X 0,Y 484.73,Z 243.524,A -85,B 0,C 180,E1 -6953.43,E2 -6953.43} C_VEL
LIN {X 0,Y 485.762,Z 223.094,A -85,B 0,C 180,E1 -6956.356,E2 -6956.356} C_VEL
LIN {X 0,Y 485.771,Z 219.542,A -85,B 0,C 180,E1 -6956.879,E2 -6956.879} C_VEL
LIN {X 0,Y 482.304,Z 204.594,A -85,B 0,C 180,E1 -6959.32,E2 -6959.32} C_VEL
LIN {X 0,Y 481.69,Z 202.108,A -85,B 0,C 180,E1 -6959.74,E2 -6959.74} C_VEL
LIN {X 0,Y 481.669,Z 202.103,A -85,B 0,C 180,E1 -6962.674,E2 -6962.674} C_VEL
LIN {X 0,Y 481.638,Z 202.112,A -85,B 0,C 180,E1 -6965.708,E2 -6965.708} C_VEL
LIN {X 0,Y 481.71,Z 202.104,A -85,B 0,C 180,E1 -6969.353,E2 -6969.353} C_VEL
LIN {X 0,Y 481.644,Z 202.116,A -85,B 0,C 180,E1 -6972.16,E2 -6972.16} C_VEL
LIN {X 0,Y 481.654,Z 202.111,A -85,B 0,C 180,E1 -6975.542,E2 -6975.542} C_VEL
LIN {X 0,Y 481.662,Z 202.106,A -85,B 0,C 180,E1 -6978.959,E2 -6978.959} C_VEL
LIN {X 0,Y 481.691,Z 202.103,A -85,B 0,C 180,E1 -6981.143,E2 -6981.143} C_VEL
LIN {X 0,Y 481.661,Z 202.105,A -85,B 0,C 180,E1 -6984.794,E2 -6984.794} C_VEL
LIN {X 0,Y 481.666,Z 202.107,A -85,B 0,C 180,E1 -6987.325,E2 -6987.325} C_VEL
LIN {X 0,Y 481.68,Z 202.106,A -85,B 0,C 180,E1 -6990.259,E2 -6990.259} C_VEL
LIN {X 0,Y 481.737,Z 202.098,A -85,B 0,C 180,E1 -6993.112,E2 -6993.112} C_VEL
LIN {X 0,Y 481.669,Z 202.11,A -85,B 0,C 180,E1 -6995.887,E2 -6995.887} C_VEL
LIN {X 0,Y 481.694,Z 202.095,A -85,B 0,C 180,E1 -6999.027,E2 -6999.027} C_VEL
LIN {X 0,Y 481.699,Z 202.105,A -85,B 0,C 180,E1 -7002.158,E2 -7002.158} C_VEL
LIN {X 0,Y 481.733,Z 202.099,A -85,B 0,C 180,E1 -7004.776,E2 -7004.776} C_VEL
LIN {X 0,Y 481.743,Z 202.098,A -85,B 0,C 180,E1 -7008.215,E2 -7008.215} C_VEL
LIN {X 0,Y 481.755,Z 202.1,A -85,B 0,C 180,E1 -7011.612,E2 -7011.612} C_VEL
LIN {X 0,Y 481.808,Z 202.09,A -85,B 0,C 180,E1 -7014.14,E2 -7014.14} C_VEL
LIN {X 0,Y 481.919,Z 202.083,A -85,B 0,C 180,E1 -7017.493,E2 -7017.493} C_VEL
LIN {X 0,Y 481.93,Z 202.073,A -85,B 0,C 180,E1 -7020,E2 -7020} C_VEL
LIN {X 0,Y 481.919,Z 202.076,A -85,B 0,C 180,E1 -7022.508,E2 -7022.508} C_VEL
LIN {X 0,Y 481.813,Z 202.091,A -85,B 0,C 180,E1 -7025.861,E2 -7025.861} C_VEL
LIN {X 0,Y 481.755,Z 202.094,A -85,B 0,C 180,E1 -7028.389,E2 -7028.389} C_VEL
LIN {X 0,Y 481.744,Z 202.098,A -85,B 0,C 180,E1 -7031.785,E2 -7031.785} C_VEL
LIN {X 0,Y 481.733,Z 202.106,A -85,B 0,C 180,E1 -7035.225,E2 -7035.225} C_VEL
LIN {X 0,Y 481.704,Z 202.106,A -85,B 0,C 180,E1 -7038.722,E2 -7038.722} C_VEL
LIN {X 0,Y 481.637,Z 202.115,A -85,B 0,C 180,E1 -7041.395,E2 -7041.395} C_VEL
LIN {X 0,Y 481.668,Z 202.105,A -85,B 0,C 180,E1 -7044.114,E2 -7044.114} C_VEL
LIN {X 0,Y 481.739,Z 202.096,A -85,B 0,C 180,E1 -7047.14,E2 -7047.14} C_VEL
LIN {X 0,Y 481.681,Z 202.106,A -85,B 0,C 180,E1 -7049.741,E2 -7049.741} C_VEL
LIN {X 0,Y 481.667,Z 202.112,A -85,B 0,C 180,E1 -7052.675,E2 -7052.675} C_VEL
LIN {X 0,Y 481.637,Z 202.111,A -85,B 0,C 180,E1 -7055.71,E2 -7055.71} C_VEL
LIN {X 0,Y 481.666,Z 202.112,A -85,B 0,C 180,E1 -7058.86,E2 -7058.86} C_VEL
LIN {X 0,Y 481.649,Z 202.107,A -85,B 0,C 180,E1 -7061.914,E2 -7061.914} C_VEL
LIN {X 0,Y 481.656,Z 202.112,A -85,B 0,C 180,E1 -7064.458,E2 -7064.458} C_VEL
LIN {X 0,Y 481.65,Z 202.11,A -85,B 0,C 180,E1 -7067.841,E2 -7067.841} C_VEL
LIN {X 0,Y 481.677,Z 202.109,A -85,B 0,C 180,E1 -7070.652,E2 -7070.652} C_VEL
LIN {X 0,Y 481.624,Z 202.114,A -85,B 0,C 180,E1 -7073.377,E2 -7073.377} C_VEL
LIN {X 0,Y 481.708,Z 202.107,A -85,B 0,C 180,E1 -7076.331,E2 -7076.331} C_VEL
LIN {X 0,Y 481.649,Z 202.114,A -85,B 0,C 180,E1 -7079.418,E2 -7079.418} C_VEL
LIN {X 0,Y 481.7,Z 202.109,A -85,B 0,C 180,E1 -7082.169,E2 -7082.169} C_VEL
LIN {X 0,Y 481.754,Z 202.257,A -85,B 0,C 180,E1 -7083.581,E2 -7083.581} C_VEL
LIN {X 0,Y 484.685,Z 215.651,A -85,B 0,C 180,E1 -7086.047,E2 -7086.047} C_VEL
LIN {X 0,Y 484.857,Z 217.051,A -85,B 0,C 180,E1 -7086.289,E2 -7086.289} C_VEL
LIN {X 0,Y 485.651,Z 219.324,A -85,B 0,C 180,E1 -7086.585,E2 -7086.585} C_VEL
LIN {X 0,Y 487.179,Z 221.975,A -85,B 0,C 180,E1 -7086.797,E2 -7086.797} C_VEL
LIN {X 0,Y 488.946,Z 225.781,A -85,B 0,C 180,E1 -7086.961,E2 -7086.961} C_VEL
LIN {X 0,Y 489.239,Z 228.795,A -85,B 0,C 180,E1 -7087.022,E2 -7087.022} C_VEL
LIN {X 0,Y 488.412,Z 231.951,A -85,B 0,C 180,E1 -7087.028,E2 -7087.028} C_VEL
LIN {X 0,Y 484.246,Z 240.493,A -85,B 0,C 180,E1 -7086.954,E2 -7086.954} C_VEL
LIN {X 0,Y 482.48,Z 248.258,A -85,B 0,C 180,E1 -7086.987,E2 -7086.987} C_VEL
LIN {X 0,Y 481.385,Z 351.579,A -85,B 0,C 180,E1 -7088.566,E2 -7088.566} C_VEL
LIN {X 0,Y 480.943,Z 385.815,A -85,B 0,C 180,E1 -7089.117,E2 -7089.117} C_VEL
LIN {X 0,Y 480.585,Z 401.032,A -85,B 0,C 180,E1 -7089.536,E2 -7089.536} C_VEL
LIN {X 0,Y 480.072,Z 414.905,A -85,B 0,C 180,E1 -7090.071,E2 -7090.071} C_VEL
LIN {X 0,Y 479.369,Z 428.202,A -85,B 0,C 180,E1 -7090.74,E2 -7090.74} C_VEL
LIN {X 0,Y 478.641,Z 441.793,A -85,B 0,C 180,E1 -7091.598,E2 -7091.598} C_VEL
LIN {X 0,Y 477.898,Z 454.287,A -85,B 0,C 180,E1 -7092.565,E2 -7092.565} C_VEL
LIN {X 0,Y 477.043,Z 466.936,A -85,B 0,C 180,E1 -7093.745,E2 -7093.745} C_VEL
LIN {X 0,Y 476.288,Z 478.4,A -85,B 0,C 180,E1 -7095.036,E2 -7095.036} C_VEL
LIN {X 0,Y 475.654,Z 488.045,A -85,B 0,C 180,E1 -7096.326,E2 -7096.326} C_VEL
LIN {X 0,Y 475.031,Z 496.792,A -85,B 0,C 180,E1 -7097.704,E2 -7097.704} C_VEL
LIN {X 0,Y 474.697,Z 504.36,A -85,B 0,C 180,E1 -7099.119,E2 -7099.119} C_VEL
LIN {X 0,Y 474.32,Z 511.031,A -85,B 0,C 180,E1 -7100.62,E2 -7100.62} C_VEL
LIN {X 0,Y 474.062,Z 517.209,A -85,B 0,C 180,E1 -7102.333,E2 -7102.333} C_VEL
LIN {X 0,Y 473.964,Z 521.979,A -85,B 0,C 180,E1 -7104.042,E2 -7104.042} C_VEL
LIN {X 0,Y 473.772,Z 525.479,A -85,B 0,C 180,E1 -7105.747,E2 -7105.747} C_VEL
LIN {X 0,Y 473.758,Z 527.793,A -85,B 0,C 180,E1 -7107.449,E2 -7107.449} C_VEL
LIN {X 0,Y 473.686,Z 528.979,A -85,B 0,C 180,E1 -7109.15,E2 -7109.15} C_VEL
LIN {X 0,Y 473.686,Z 528.996,A -85,B 0,C 180,E1 -7110.85,E2 -7110.85} C_VEL
LIN {X 0,Y 473.758,Z 527.881,A -85,B 0,C 180,E1 -7112.551,E2 -7112.551} C_VEL
LIN {X 0,Y 473.77,Z 525.636,A -85,B 0,C 180,E1 -7114.253,E2 -7114.253} C_VEL
LIN {X 0,Y 473.941,Z 522.201,A -85,B 0,C 180,E1 -7115.958,E2 -7115.958} C_VEL
LIN {X 0,Y 474.061,Z 517.503,A -85,B 0,C 180,E1 -7117.667,E2 -7117.667} C_VEL
LIN {X 0,Y 474.294,Z 511.413,A -85,B 0,C 180,E1 -7119.381,E2 -7119.381} C_VEL
LIN {X 0,Y 474.785,Z 503.739,A -85,B 0,C 180,E1 -7121.094,E2 -7121.094} C_VEL
LIN {X 0,Y 475.142,Z 496.043,A -85,B 0,C 180,E1 -7122.517,E2 -7122.517} C_VEL
LIN {X 0,Y 475.83,Z 485.703,A -85,B 0,C 180,E1 -7124.105,E2 -7124.105} C_VEL
LIN {X 0,Y 476.492,Z 475.593,A -85,B 0,C 180,E1 -7125.396,E2 -7125.396} C_VEL
LIN {X 0,Y 477.175,Z 465.429,A -85,B 0,C 180,E1 -7126.496,E2 -7126.496} C_VEL
LIN {X 0,Y 477.975,Z 452.771,A -85,B 0,C 180,E1 -7127.653,E2 -7127.653} C_VEL
LIN {X 0,Y 478.78,Z 439.944,A -85,B 0,C 180,E1 -7128.618,E2 -7128.618} C_VEL
LIN {X 0,Y 479.486,Z 425.876,A -85,B 0,C 180,E1 -7129.478,E2 -7129.478} C_VEL
LIN {X 0,Y 480.204,Z 410.756,A -85,B 0,C 180,E1 -7130.193,E2 -7130.193} C_VEL
LIN {X 0,Y 480.683,Z 395.645,A -85,B 0,C 180,E1 -7130.723,E2 -7130.723} C_VEL
LIN {X 0,Y 481.037,Z 381.858,A -85,B 0,C 180,E1 -7131.052,E2 -7131.052} C_VEL
LIN {X 0,Y 482.436,Z 253.492,A -85,B 0,C 180,E1 -7133.024,E2 -7133.024} C_VEL
LIN {X 0,Y 482.51,Z 238.488,A -85,B 0,C 180,E1 -7133.258,E2 -7133.258} C_VEL
LIN {X 0,Y 478.11,Z 219.337,A -85,B 0,C 180,E1 -7133.805,E2 -7133.805} C_VEL
LIN {X 0,Y 476.509,Z 211.019,A -85,B 0,C 180,E1 -7135.322,E2 -7135.322} C_VEL
LIN {X 0,Y 474.705,Z 202.984,A -85,B 0,C 180,E1 -7136.872,E2 -7136.872} C_VEL
LIN {X 0,Y 474.604,Z 202.991,A -85,B 0,C 180,E1 -7140.229,E2 -7140.229} C_VEL
LIN {X 0,Y 474.641,Z 202.992,A -85,B 0,C 180,E1 -7143.219,E2 -7143.219} C_VEL
LIN {X 0,Y 474.589,Z 202.991,A -85,B 0,C 180,E1 -7146.323,E2 -7146.323} C_VEL
LIN {X 0,Y 474.624,Z 202.987,A -85,B 0,C 180,E1 -7149.647,E2 -7149.647} C_VEL
LIN {X 0,Y 474.631,Z 202.987,A -85,B 0,C 180,E1 -7152.931,E2 -7152.931} C_VEL
LIN {X 0,Y 474.605,Z 202.988,A -85,B 0,C 180,E1 -7155.894,E2 -7155.894} C_VEL
LIN {X 0,Y 474.636,Z 202.985,A -85,B 0,C 180,E1 -7159.038,E2 -7159.038} C_VEL
LIN {X 0,Y 474.609,Z 202.981,A -85,B 0,C 180,E1 -7161.703,E2 -7161.703} C_VEL
LIN {X 0,Y 474.624,Z 202.986,A -85,B 0,C 180,E1 -7164.725,E2 -7164.725} C_VEL
LIN {X 0,Y 474.63,Z 202.975,A -85,B 0,C 180,E1 -7167.787,E2 -7167.787} C_VEL
LIN {X 0,Y 474.625,Z 202.987,A -85,B 0,C 180,E1 -7170.882,E2 -7170.882} C_VEL
LIN {X 0,Y 474.652,Z 202.98,A -85,B 0,C 180,E1 -7173.628,E2 -7173.628} C_VEL
LIN {X 0,Y 474.628,Z 202.988,A -85,B 0,C 180,E1 -7176.641,E2 -7176.641} C_VEL
LIN {X 0,Y 474.648,Z 202.982,A -85,B 0,C 180,E1 -7180.089,E2 -7180.089} C_VEL
LIN {X 0,Y 474.643,Z 202.986,A -85,B 0,C 180,E1 -7182.774,E2 -7182.774} C_VEL
LIN {X 0,Y 474.64,Z 202.98,A -85,B 0,C 180,E1 -7185.421,E2 -7185.421} C_VEL
LIN {X 0,Y 474.696,Z 202.976,A -85,B 0,C 180,E1 -7188.037,E2 -7188.037} C_VEL
LIN {X 0,Y 474.719,Z 202.973,A -85,B 0,C 180,E1 -7191.486,E2 -7191.486} C_VEL
LIN {X 0,Y 474.77,Z 202.966,A -85,B 0,C 180,E1 -7194.052,E2 -7194.052} C_VEL
LIN {X 0,Y 474.885,Z 202.953,A -85,B 0,C 180,E1 -7197.455,E2 -7197.455} C_VEL
LIN {X 0,Y 474.868,Z 202.96,A -85,B 0,C 180,E1 -7200.848,E2 -7200.848} C_VEL
LIN {X 0,Y 474.885,Z 202.959,A -85,B 0,C 180,E1 -7202.545,E2 -7202.545} C_VEL
LIN {X 0,Y 474.77,Z 202.968,A -85,B 0,C 180,E1 -7205.948,E2 -7205.948} C_VEL
LIN {X 0,Y 474.72,Z 202.976,A -85,B 0,C 180,E1 -7208.514,E2 -7208.514} C_VEL
LIN {X 0,Y 474.696,Z 202.978,A -85,B 0,C 180,E1 -7211.963,E2 -7211.963} C_VEL
LIN {X 0,Y 474.691,Z 202.978,A -85,B 0,C 180,E1 -7215.456,E2 -7215.456} C_VEL
LIN {X 0,Y 474.657,Z 202.984,A -85,B 0,C 180,E1 -7219.01,E2 -7219.01} C_VEL
LIN {X 0,Y 474.581,Z 202.989,A -85,B 0,C 180,E1 -7221.729,E2 -7221.729} C_VEL
LIN {X 0,Y 474.65,Z 202.985,A -85,B 0,C 180,E1 -7224.493,E2 -7224.493} C_VEL
LIN {X 0,Y 474.691,Z 202.977,A -85,B 0,C 180,E1 -7227.339,E2 -7227.339} C_VEL
LIN {X 0,Y 474.602,Z 202.99,A -85,B 0,C 180,E1 -7230.812,E2 -7230.812} C_VEL
LIN {X 0,Y 474.631,Z 202.987,A -85,B 0,C 180,E1 -7233.985,E2 -7233.985} C_VEL
LIN {X 0,Y 474.568,Z 202.992,A -85,B 0,C 180,E1 -7236.9,E2 -7236.9} C_VEL
LIN {X 0,Y 474.621,Z 202.985,A -85,B 0,C 180,E1 -7239.648,E2 -7239.648} C_VEL
LIN {X 0,Y 474.609,Z 202.988,A -85,B 0,C 180,E1 -7242.935,E2 -7242.935} C_VEL
LIN {X 0,Y 474.604,Z 202.994,A -85,B 0,C 180,E1 -7245.896,E2 -7245.896} C_VEL
LIN {X 0,Y 474.637,Z 202.984,A -85,B 0,C 180,E1 -7249.039,E2 -7249.039} C_VEL
LIN {X 0,Y 474.612,Z 202.99,A -85,B 0,C 180,E1 -7251.704,E2 -7251.704} C_VEL
LIN {X 0,Y 474.625,Z 202.987,A -85,B 0,C 180,E1 -7254.727,E2 -7254.727} C_VEL
LIN {X 0,Y 474.633,Z 202.99,A -85,B 0,C 180,E1 -7257.788,E2 -7257.788} C_VEL
LIN {X 0,Y 474.676,Z 203.113,A -85,B 0,C 180,E1 -7259.96,E2 -7259.96} C_VEL
LIN {X 0,Y 478.246,Z 217.916,A -85,B 0,C 180,E1 -7262.448,E2 -7262.448} C_VEL
LIN {X 0,Y 479.058,Z 222.313,A -85,B 0,C 180,E1 -7263.155,E2 -7263.155} C_VEL
LIN {X 0,Y 477.935,Z 243.39,A -85,B 0,C 180,E1 -7266.224,E2 -7266.224} C_VEL
LIN {X 0,Y 482.436,Z 267.104,A -85,B 0,C 180,E1 -7266.839,E2 -7266.839} C_VEL
LIN {X 0,Y 480.808,Z 410.383,A -85,B 0,C 180,E1 -7269.044,E2 -7269.044} C_VEL
LIN {X 0,Y 480.262,Z 426.409,A -85,B 0,C 180,E1 -7269.473,E2 -7269.473} C_VEL
LIN {X 0,Y 479.688,Z 441.446,A -85,B 0,C 180,E1 -7270.058,E2 -7270.058} C_VEL
LIN {X 0,Y 478.978,Z 454.629,A -85,B 0,C 180,E1 -7270.723,E2 -7270.723} C_VEL
LIN {X 0,Y 478.256,Z 468.14,A -85,B 0,C 180,E1 -7271.583,E2 -7271.583} C_VEL
LIN {X 0,Y 477.319,Z 481.894,A -85,B 0,C 180,E1 -7272.653,E2 -7272.653} C_VEL
LIN {X 0,Y 476.573,Z 494.351,A -85,B 0,C 180,E1 -7273.839,E2 -7273.839} C_VEL
LIN {X 0,Y 475.86,Z 504.795,A -85,B 0,C 180,E1 -7275.022,E2 -7275.022} C_VEL
LIN {X 0,Y 475.256,Z 514.494,A -85,B 0,C 180,E1 -7276.314,E2 -7276.314} C_VEL
LIN {X 0,Y 474.72,Z 523.406,A -85,B 0,C 180,E1 -7277.714,E2 -7277.714} C_VEL
LIN {X 0,Y 474.389,Z 531.965,A -85,B 0,C 180,E1 -7279.328,E2 -7279.328} C_VEL
LIN {X 0,Y 474.045,Z 539.378,A -85,B 0,C 180,E1 -7281.045,E2 -7281.045} C_VEL
LIN {X 0,Y 473.904,Z 545.262,A -85,B 0,C 180,E1 -7282.758,E2 -7282.758} C_VEL
LIN {X 0,Y 473.789,Z 548.758,A -85,B 0,C 180,E1 -7284.04,E2 -7284.04} C_VEL
LIN {X 0,Y 473.684,Z 552.291,A -85,B 0,C 180,E1 -7285.746,E2 -7285.746} C_VEL
LIN {X 0,Y 473.734,Z 554.619,A -85,B 0,C 180,E1 -7287.449,E2 -7287.449} C_VEL
LIN {X 0,Y 473.686,Z 555.788,A -85,B 0,C 180,E1 -7289.15,E2 -7289.15} C_VEL
LIN {X 0,Y 473.686,Z 555.787,A -85,B 0,C 180,E1 -7290.85,E2 -7290.85} C_VEL
LIN {X 0,Y 473.734,Z 554.614,A -85,B 0,C 180,E1 -7292.551,E2 -7292.551} C_VEL
LIN {X 0,Y 473.684,Z 552.286,A -85,B 0,C 180,E1 -7294.254,E2 -7294.254} C_VEL
LIN {X 0,Y 473.81,Z 548.759,A -85,B 0,C 180,E1 -7295.96,E2 -7295.96} C_VEL
LIN {X 0,Y 473.907,Z 543.937,A -85,B 0,C 180,E1 -7297.67,E2 -7297.67} C_VEL
LIN {X 0,Y 474.094,Z 537.693,A -85,B 0,C 180,E1 -7299.385,E2 -7299.385} C_VEL
LIN {X 0,Y 474.511,Z 529.854,A -85,B 0,C 180,E1 -7301.101,E2 -7301.101} C_VEL
LIN {X 0,Y 474.854,Z 521.294,A -85,B 0,C 180,E1 -7302.644,E2 -7302.644} C_VEL
LIN {X 0,Y 475.452,Z 511.474,A -85,B 0,C 180,E1 -7304.116,E2 -7304.116} C_VEL
LIN {X 0,Y 476.091,Z 501.206,A -85,B 0,C 180,E1 -7305.409,E2 -7305.409} C_VEL
LIN {X 0,Y 476.899,Z 489.12,A -85,B 0,C 180,E1 -7306.686,E2 -7306.686} C_VEL
LIN {X 0,Y 477.649,Z 476.704,A -85,B 0,C 180,E1 -7307.776,E2 -7307.776} C_VEL
LIN {X 0,Y 478.508,Z 463.356,A -85,B 0,C 180,E1 -7308.74,E2 -7308.74} C_VEL
LIN {X 0,Y 479.298,Z 448.626,A -85,B 0,C 180,E1 -7309.598,E2 -7309.598} C_VEL
LIN {X 0,Y 480.003,Z 434.065,A -85,B 0,C 180,E1 -7310.25,E2 -7310.25} C_VEL
LIN {X 0,Y 480.526,Z 419.095,A -85,B 0,C 180,E1 -7310.745,E2 -7310.745} C_VEL
LIN {X 0,Y 480.935,Z 404.456,A -85,B 0,C 180,E1 -7311.062,E2 -7311.062} C_VEL
LIN {X 0,Y 482.436,Z 266.978,A -85,B 0,C 180,E1 -7313.161,E2 -7313.161} C_VEL
LIN {X 0,Y 477.922,Z 243.373,A -85,B 0,C 180,E1 -7313.775,E2 -7313.775} C_VEL
LIN {X 0,Y 478.994,Z 223.374,A -85,B 0,C 180,E1 -7316.686,E2 -7316.686} C_VEL
LIN {X 0,Y 478.592,Z 219.413,A -85,B 0,C 180,E1 -7317.304,E2 -7317.304} C_VEL
LIN {X 0,Y 475.131,Z 205.065,A -85,B 0,C 180,E1 -7319.703,E2 -7319.703} C_VEL
LIN {X 0,Y 474.616,Z 202.988,A -85,B 0,C 180,E1 -7320.075,E2 -7320.075} C_VEL
LIN {X 0,Y 474.64,Z 202.976,A -85,B 0,C 180,E1 -7323.219,E2 -7323.219} C_VEL
LIN {X 0,Y 474.588,Z 202.993,A -85,B 0,C 180,E1 -7326.323,E2 -7326.323} C_VEL
LIN {X 0,Y 474.646,Z 202.987,A -85,B 0,C 180,E1 -7329.65,E2 -7329.65} C_VEL
LIN {X 0,Y 474.61,Z 202.986,A -85,B 0,C 180,E1 -7332.934,E2 -7332.934} C_VEL
LIN {X 0,Y 474.604,Z 202.993,A -85,B 0,C 180,E1 -7335.895,E2 -7335.895} C_VEL
LIN {X 0,Y 474.635,Z 202.982,A -85,B 0,C 180,E1 -7339.038,E2 -7339.038} C_VEL
LIN {X 0,Y 474.61,Z 202.989,A -85,B 0,C 180,E1 -7341.702,E2 -7341.702} C_VEL
LIN {X 0,Y 474.623,Z 202.982,A -85,B 0,C 180,E1 -7344.726,E2 -7344.726} C_VEL
LIN {X 0,Y 474.63,Z 202.987,A -85,B 0,C 180,E1 -7347.787,E2 -7347.787} C_VEL
LIN {X 0,Y 474.624,Z 202.983,A -85,B 0,C 180,E1 -7350.882,E2 -7350.882} C_VEL
LIN {X 0,Y 474.652,Z 202.985,A -85,B 0,C 180,E1 -7353.628,E2 -7353.628} C_VEL
LIN {X 0,Y 474.627,Z 202.981,A -85,B 0,C 180,E1 -7356.641,E2 -7356.641} C_VEL
LIN {X 0,Y 474.648,Z 202.983,A -85,B 0,C 180,E1 -7360.089,E2 -7360.089} C_VEL
LIN {X 0,Y 474.642,Z 202.982,A -85,B 0,C 180,E1 -7362.774,E2 -7362.774} C_VEL
LIN {X 0,Y 474.64,Z 202.988,A -85,B 0,C 180,E1 -7365.421,E2 -7365.421} C_VEL
LIN {X 0,Y 474.696,Z 202.977,A -85,B 0,C 180,E1 -7368.037,E2 -7368.037} C_VEL
LIN {X 0,Y 474.72,Z 202.976,A -85,B 0,C 180,E1 -7371.486,E2 -7371.486} C_VEL
LIN {X 0,Y 474.77,Z 202.968,A -85,B 0,C 180,E1 -7374.052,E2 -7374.052} C_VEL
LIN {X 0,Y 474.885,Z 202.96,A -85,B 0,C 180,E1 -7377.455,E2 -7377.455} C_VEL
LIN {X 0,Y 474.868,Z 202.953,A -85,B 0,C 180,E1 -7380.848,E2 -7380.848} C_VEL
LIN {X 0,Y 474.886,Z 202.953,A -85,B 0,C 180,E1 -7382.545,E2 -7382.545} C_VEL
LIN {X 0,Y 474.775,Z 202.967,A -85,B 0,C 180,E1 -7385.948,E2 -7385.948} C_VEL
LIN {X 0,Y 474.72,Z 202.97,A -85,B 0,C 180,E1 -7388.514,E2 -7388.514} C_VEL
LIN {X 0,Y 474.697,Z 202.974,A -85,B 0,C 180,E1 -7391.963,E2 -7391.963} C_VEL
LIN {X 0,Y 474.691,Z 202.979,A -85,B 0,C 180,E1 -7395.456,E2 -7395.456} C_VEL
LIN {X 0,Y 474.656,Z 202.987,A -85,B 0,C 180,E1 -7399.011,E2 -7399.011} C_VEL
LIN {X 0,Y 474.58,Z 202.991,A -85,B 0,C 180,E1 -7401.729,E2 -7401.729} C_VEL
LIN {X 0,Y 474.651,Z 202.981,A -85,B 0,C 180,E1 -7404.493,E2 -7404.493} C_VEL
LIN {X 0,Y 474.692,Z 202.978,A -85,B 0,C 180,E1 -7407.339,E2 -7407.339} C_VEL
LIN {X 0,Y 474.603,Z 202.992,A -85,B 0,C 180,E1 -7410.812,E2 -7410.812} C_VEL
LIN {X 0,Y 474.632,Z 202.981,A -85,B 0,C 180,E1 -7413.985,E2 -7413.985} C_VEL
LIN {X 0,Y 474.569,Z 202.995,A -85,B 0,C 180,E1 -7416.901,E2 -7416.901} C_VEL
LIN {X 0,Y 474.622,Z 202.983,A -85,B 0,C 180,E1 -7419.648,E2 -7419.648} C_VEL
LIN {X 0,Y 474.635,Z 202.989,A -85,B 0,C 180,E1 -7422.932,E2 -7422.932} C_VEL
LIN {X 0,Y 474.611,Z 202.987,A -85,B 0,C 180,E1 -7425.897,E2 -7425.897} C_VEL
LIN {X 0,Y 474.629,Z 202.99,A -85,B 0,C 180,E1 -7429.041,E2 -7429.041} C_VEL
LIN {X 0,Y 474.607,Z 202.987,A -85,B 0,C 180,E1 -7431.705,E2 -7431.705} C_VEL
LIN {X 0,Y 474.622,Z 202.99,A -85,B 0,C 180,E1 -7434.726,E2 -7434.726} C_VEL
LIN {X 0,Y 474.634,Z 202.987,A -85,B 0,C 180,E1 -7437.788,E2 -7437.788} C_VEL
LIN {X 0,Y 474.623,Z 202.99,A -85,B 0,C 180,E1 -7440.885,E2 -7440.885} C_VEL
LIN {X 0,Y 474.732,Z 203.12,A -85,B 0,C 180,E1 -7443.278,E2 -7443.278} C_VEL
LIN {X 0,Y 477.698,Z 216.633,A -85,B 0,C 180,E1 -7445.805,E2 -7445.805} C_VEL
LIN {X 0,Y 478.112,Z 219.59,A -85,B 0,C 180,E1 -7446.302,E2 -7446.302} C_VEL
LIN {X 0,Y 482.582,Z 239.036,A -85,B 0,C 180,E1 -7446.846,E2 -7446.846} C_VEL
LIN {X 0,Y 482.48,Z 248.258,A -85,B 0,C 180,E1 -7446.987,E2 -7446.987} C_VEL
LIN {X 0,Y 481.815,Z 254.113,A -85,B 0,C 180,E1 -7447.046,E2 -7447.046} C_VEL
LIN {X 0,Y 476.269,Z 273.184,A -85,B 0,C 180,E1 -7447.067,E2 -7447.067} C_VEL
LIN {X 0,Y 475.647,Z 279.036,A -85,B 0,C 180,E1 -7447.129,E2 -7447.129} C_VEL
LIN {X 0,Y 474.385,Z 385.004,A -85,B 0,C 180,E1 -7448.789,E2 -7448.789} C_VEL
LIN {X 0,Y 474.015,Z 400.38,A -85,B 0,C 180,E1 -7449.207,E2 -7449.207} C_VEL
